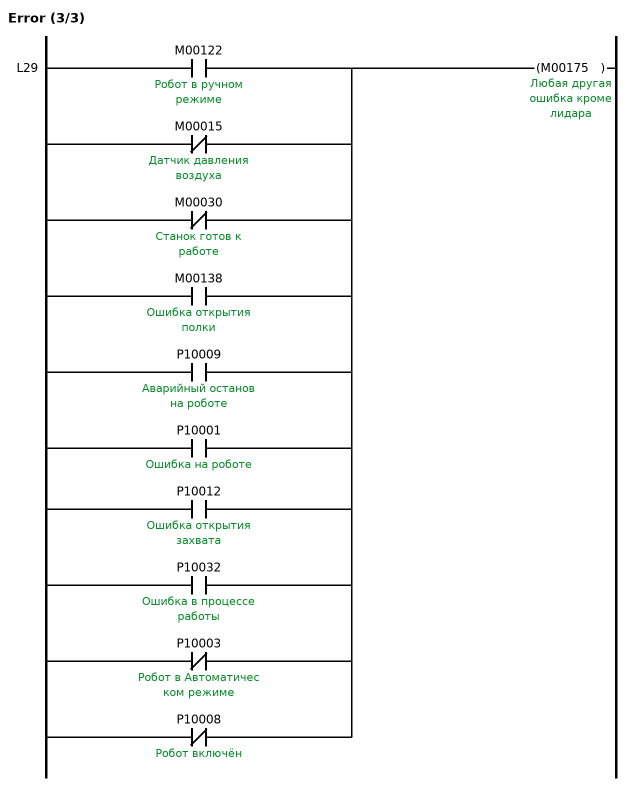
[picture p24: Error rungs L29-L29]
; L29
LOAD      M00122	// Робот в ручном режиме
OR NOT    M00015	// Датчик давления воздуха
OR NOT    M00030	// Станок готов к работе
OR        M00138	// Ошибка открытия полки
OR        P10009	// Аварийный останов на роботе
OR        P10001	// Ошибка на роботе
OR        P10012	// Ошибка открытия захвата
OR        P10032	// Ошибка в процессе работы
OR NOT    P10003	// Робот в Автоматическом режиме
OR NOT    P10008	// Робот включён
OUT       M00175	// Любая другая ошибка кроме лидара

PROGRAM Initialization (task: Scan Program)

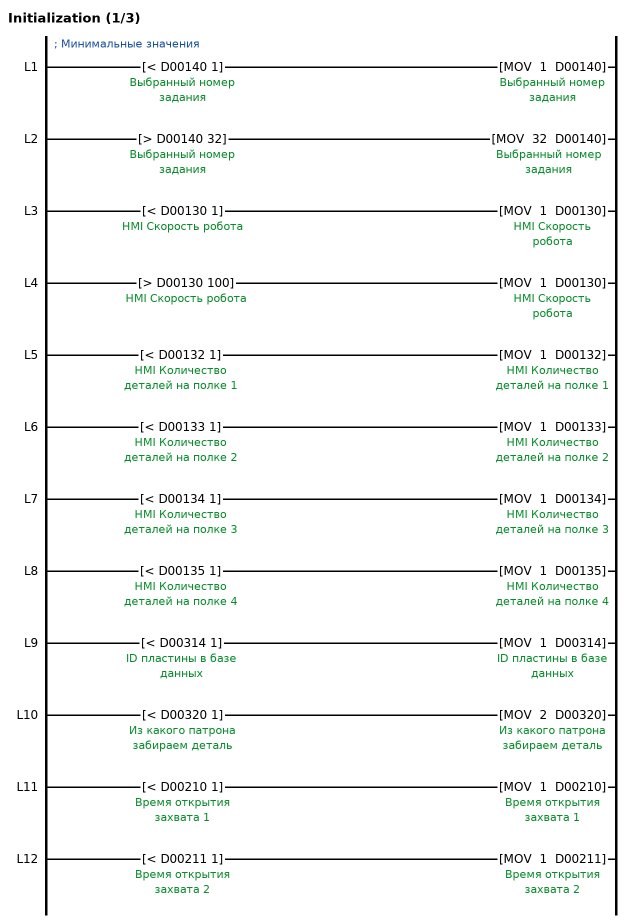
// Минимальные значения
; L1
LOAD<     D00140 1	// Выбранный номер задания
MOV       1 D00140	// Выбранный номер задания
; L2
LOAD>     D00140 32	// Выбранный номер задания
MOV       32 D00140	// Выбранный номер задания
; L3
LOAD<     D00130 1	// HMI Скорость робота
MOV       1 D00130	// HMI Скорость робота
; L4
LOAD>     D00130 100	// HMI Скорость робота
MOV       1 D00130	// HMI Скорость робота
; L5
LOAD<     D00132 1	// HMI Количество деталей на полке 1
MOV       1 D00132	// HMI Количество деталей на полке 1
; L6
LOAD<     D00133 1	// HMI Количество деталей на полке 2
MOV       1 D00133	// HMI Количество деталей на полке 2
; L7
LOAD<     D00134 1	// HMI Количество деталей на полке 3
MOV       1 D00134	// HMI Количество деталей на полке 3
; L8
LOAD<     D00135 1	// HMI Количество деталей на полке 4
MOV       1 D00135	// HMI Количество деталей на полке 4
; L9
LOAD<     D00314 1	// ID пластины в базе данных
MOV       1 D00314	// ID пластины в базе данных
; L10
LOAD<     D00320 1	// Из какого патрона забираем деталь
MOV       2 D00320	// Из какого патрона забираем деталь
; L11
LOAD<     D00210 1	// Время открытия захвата 1
MOV       1 D00210	// Время открытия захвата 1
; L12
LOAD<     D00211 1	// Время открытия захвата 2
MOV       1 D00211	// Время открытия захвата 2

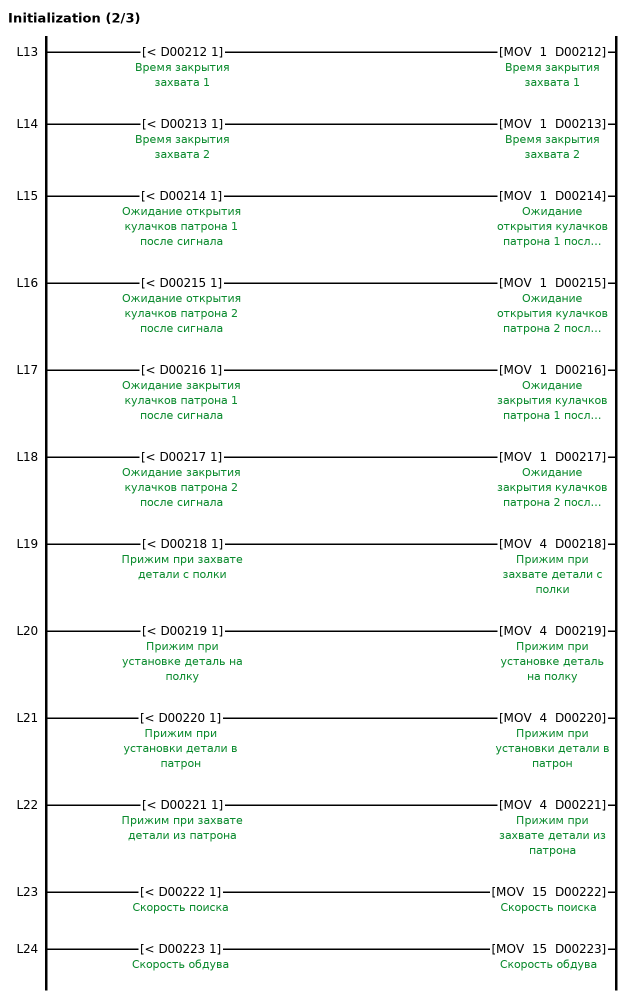
; L13
LOAD<     D00212 1	// Время закрытия захвата 1
MOV       1 D00212	// Время закрытия захвата 1
; L14
LOAD<     D00213 1	// Время закрытия захвата 2
MOV       1 D00213	// Время закрытия захвата 2
; L15
LOAD<     D00214 1	// Ожидание открытия кулачков патрона 1 после сигнала 
MOV       1 D00214	// Ожидание открытия кулачков патрона 1 после сигнала 
; L16
LOAD<     D00215 1	// Ожидание открытия кулачков патрона 2 после сигнала 
MOV       1 D00215	// Ожидание открытия кулачков патрона 2 после сигнала 
; L17
LOAD<     D00216 1	// Ожидание закрытия кулачков патрона 1 после сигнала 
MOV       1 D00216	// Ожидание закрытия кулачков патрона 1 после сигнала 
; L18
LOAD<     D00217 1	// Ожидание закрытия кулачков патрона 2 после сигнала 
MOV       1 D00217	// Ожидание закрытия кулачков патрона 2 после сигнала 
; L19
LOAD<     D00218 1	// Прижим при захвате детали с полки
MOV       4 D00218	// Прижим при захвате детали с полки
; L20
LOAD<     D00219 1	// Прижим при установке деталь на полку
MOV       4 D00219	// Прижим при установке деталь на полку
; L21
LOAD<     D00220 1	// Прижим при установки детали в патрон
MOV       4 D00220	// Прижим при установки детали в патрон
; L22
LOAD<     D00221 1	// Прижим при захвате детали из патрона
MOV       4 D00221	// Прижим при захвате детали из патрона
; L23
LOAD<     D00222 1	// Скорость поиска
MOV       15 D00222	// Скорость поиска
; L24
LOAD<     D00223 1	// Скорость обдува
MOV       15 D00223	// Скорость обдува

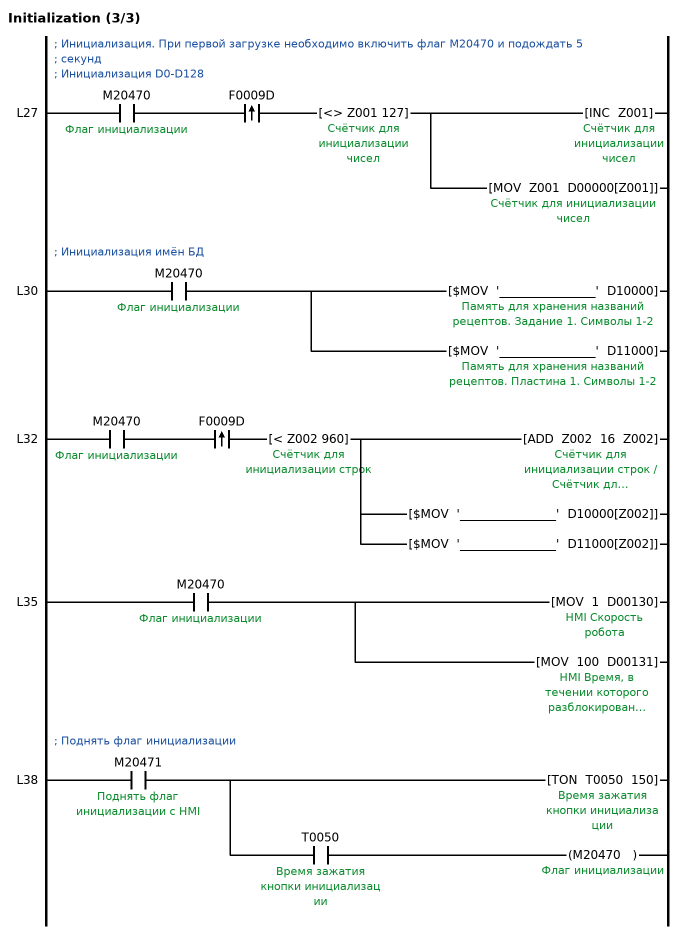
// Инициализация. При первой загрузке необходимо включить флаг M20470 и подождать 5 секунд
// Инициализация D0-D128
; L27
LOAD      M20470	// Флаг инициализации
ANDP      F0009D
AND<>     Z001 127	// Счётчик для инициализации чисел
INC       Z001	// Счётчик для инициализации чисел
MOV       Z001 D00000[Z001]	// Счётчик для инициализации чисел
// Инициализация имён БД
; L30
LOAD      M20470	// Флаг инициализации
$MOV      '________________' D10000	// Память для хранения названий рецептов. Задание 1. Символы 1-2
$MOV      '________________' D11000	// Память для хранения названий рецептов. Пластина 1. Символы 1-2
; L32
LOAD      M20470	// Флаг инициализации
ANDP      F0009D
AND<      Z002 960	// Счётчик для инициализации строк
ADD       Z002 16 Z002	// Счётчик для инициализации строк / Счётчик для инициализации строк
$MOV      '________________' D10000[Z002]
$MOV      '________________' D11000[Z002]
; L35
LOAD      M20470	// Флаг инициализации
MOV       1 D00130	// HMI Скорость робота
MOV       100 D00131	// HMI Время, в течении которого разблокирована полка после нажатия кнопки
// Поднять флаг инициализации
; L38
LOAD      M20471	// Поднять флаг инициализации с HMI
TON       T0050 150	// Время зажатия кнопки инициализации
AND       T0050	// Время зажатия кнопки инициализации
OUT       M20470	// Флаг инициализации

PROGRAM Shelves (task: Scan Program)

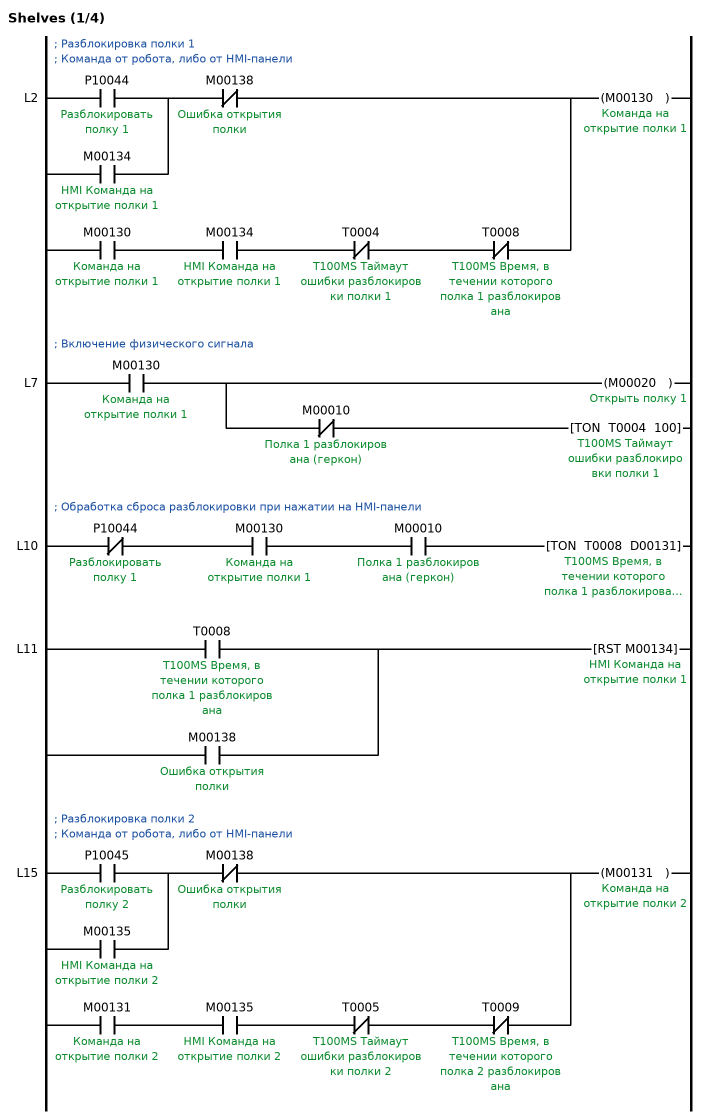
// Разблокировка полки 1
// Команда от робота, либо от HMI-панели
; L2
LOAD      P10044	// Разблокировать полку 1
OR        M00134	// HMI Команда на открытие полки 1
AND NOT   M00138	// Ошибка открытия полки
LOAD      M00130	// Команда на открытие полки 1
AND       M00134	// HMI Команда на открытие полки 1
AND NOT   T0004	// T100MS Таймаут ошибки разблокировки полки 1
AND NOT   T0008	// T100MS Время, в течении которого полка 1 разблокирована
OR LOAD
OUT       M00130	// Команда на открытие полки 1
// Включение физического сигнала
; L7
LOAD      M00130	// Команда на открытие полки 1
OUT       M00020	// Открыть полку 1
AND NOT   M00010	// Полка 1 разблокирована (геркон)
TON       T0004 100	// T100MS Таймаут ошибки разблокировки полки 1
// Обработка сброса разблокировки при нажатии на HMI-панели
; L10
LOAD NOT  P10044	// Разблокировать полку 1
AND       M00130	// Команда на открытие полки 1
AND       M00010	// Полка 1 разблокирована (геркон)
TON       T0008 D00131	// T100MS Время, в течении которого полка 1 разблокирована / HMI Время, в течении которого разблокирована полка после нажатия кнопки
; L11
LOAD      T0008	// T100MS Время, в течении которого полка 1 разблокирована
OR        M00138	// Ошибка открытия полки
RST       M00134	// HMI Команда на открытие полки 1
// Разблокировка полки 2
// Команда от робота, либо от HMI-панели
; L15
LOAD      P10045	// Разблокировать полку 2
OR        M00135	// HMI Команда на открытие полки 2
AND NOT   M00138	// Ошибка открытия полки
LOAD      M00131	// Команда на открытие полки 2
AND       M00135	// HMI Команда на открытие полки 2
AND NOT   T0005	// T100MS Таймаут ошибки разблокировки полки 2
AND NOT   T0009	// T100MS Время, в течении которого полка 2 разблокирована
OR LOAD
OUT       M00131	// Команда на открытие полки 2

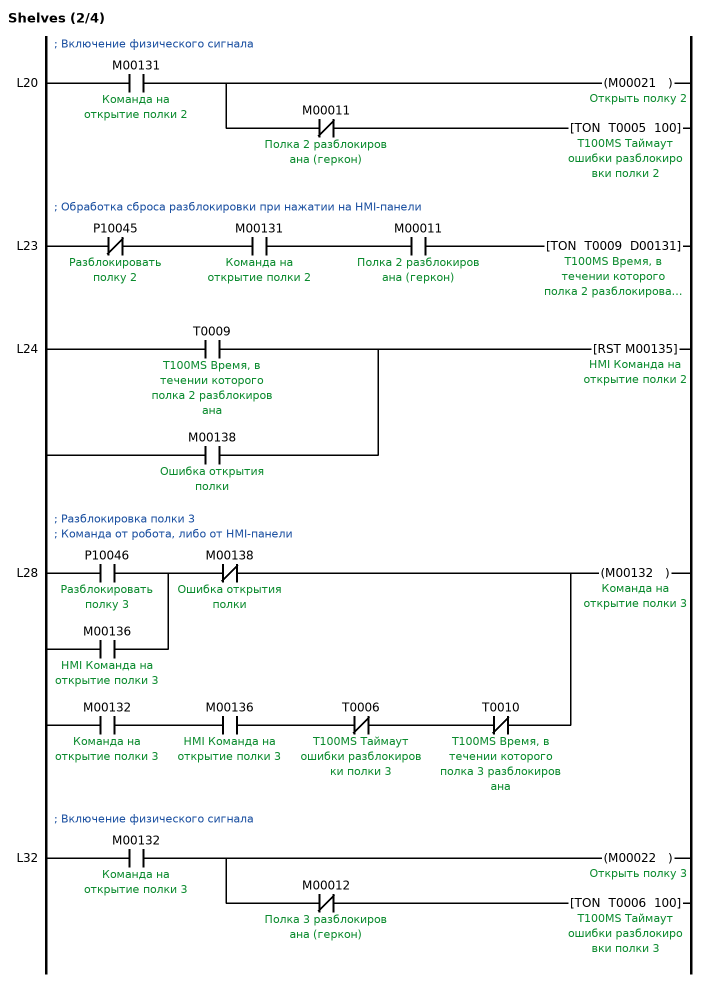
// Включение физического сигнала
; L20
LOAD      M00131	// Команда на открытие полки 2
OUT       M00021	// Открыть полку 2
AND NOT   M00011	// Полка 2 разблокирована (геркон)
TON       T0005 100	// T100MS Таймаут ошибки разблокировки полки 2
// Обработка сброса разблокировки при нажатии на HMI-панели
; L23
LOAD NOT  P10045	// Разблокировать полку 2
AND       M00131	// Команда на открытие полки 2
AND       M00011	// Полка 2 разблокирована (геркон)
TON       T0009 D00131	// T100MS Время, в течении которого полка 2 разблокирована / HMI Время, в течении которого разблокирована полка после нажатия кнопки
; L24
LOAD      T0009	// T100MS Время, в течении которого полка 2 разблокирована
OR        M00138	// Ошибка открытия полки
RST       M00135	// HMI Команда на открытие полки 2
// Разблокировка полки 3
// Команда от робота, либо от HMI-панели
; L28
LOAD      P10046	// Разблокировать полку 3
OR        M00136	// HMI Команда на открытие полки 3
AND NOT   M00138	// Ошибка открытия полки
LOAD      M00132	// Команда на открытие полки 3
AND       M00136	// HMI Команда на открытие полки 3
AND NOT   T0006	// T100MS Таймаут ошибки разблокировки полки 3
AND NOT   T0010	// T100MS Время, в течении которого полка 3 разблокирована
OR LOAD
OUT       M00132	// Команда на открытие полки 3
// Включение физического сигнала
; L32
LOAD      M00132	// Команда на открытие полки 3
OUT       M00022	// Открыть полку 3
AND NOT   M00012	// Полка 3 разблокирована (геркон)
TON       T0006 100	// T100MS Таймаут ошибки разблокировки полки 3

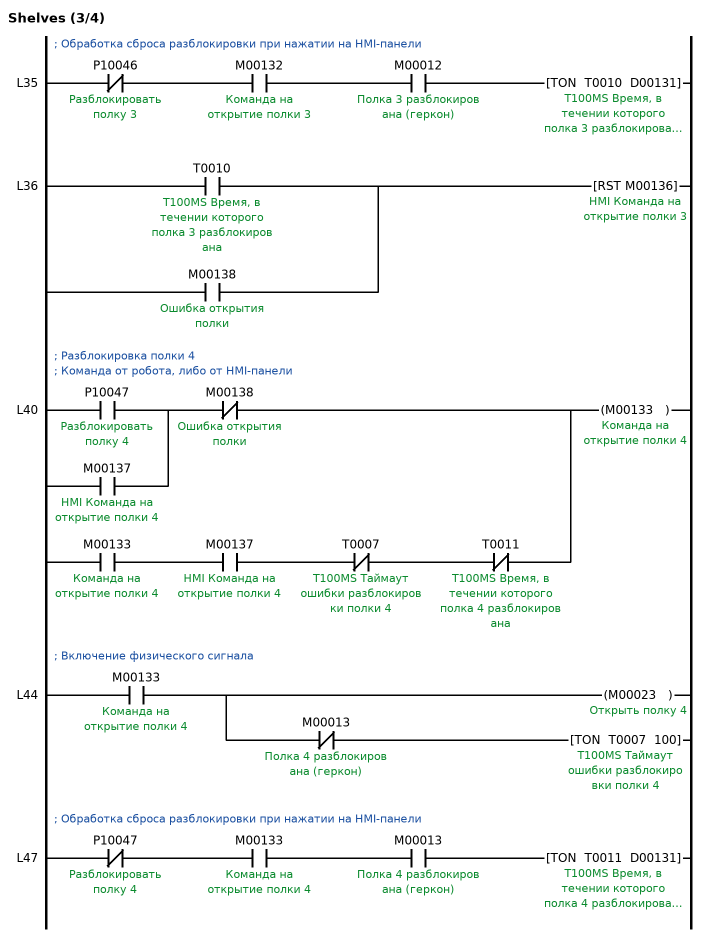
// Обработка сброса разблокировки при нажатии на HMI-панели
; L35
LOAD NOT  P10046	// Разблокировать полку 3
AND       M00132	// Команда на открытие полки 3
AND       M00012	// Полка 3 разблокирована (геркон)
TON       T0010 D00131	// T100MS Время, в течении которого полка 3 разблокирована / HMI Время, в течении которого разблокирована полка после нажатия кнопки
; L36
LOAD      T0010	// T100MS Время, в течении которого полка 3 разблокирована
OR        M00138	// Ошибка открытия полки
RST       M00136	// HMI Команда на открытие полки 3
// Разблокировка полки 4
// Команда от робота, либо от HMI-панели
; L40
LOAD      P10047	// Разблокировать полку 4
OR        M00137	// HMI Команда на открытие полки 4
AND NOT   M00138	// Ошибка открытия полки
LOAD      M00133	// Команда на открытие полки 4
AND       M00137	// HMI Команда на открытие полки 4
AND NOT   T0007	// T100MS Таймаут ошибки разблокировки полки 4
AND NOT   T0011	// T100MS Время, в течении которого полка 4 разблокирована
OR LOAD
OUT       M00133	// Команда на открытие полки 4
// Включение физического сигнала
; L44
LOAD      M00133	// Команда на открытие полки 4
OUT       M00023	// Открыть полку 4
AND NOT   M00013	// Полка 4 разблокирована (геркон)
TON       T0007 100	// T100MS Таймаут ошибки разблокировки полки 4
// Обработка сброса разблокировки при нажатии на HMI-панели
; L47
LOAD NOT  P10047	// Разблокировать полку 4
AND       M00133	// Команда на открытие полки 4
AND       M00013	// Полка 4 разблокирована (геркон)
TON       T0011 D00131	// T100MS Время, в течении которого полка 4 разблокирована / HMI Время, в течении которого разблокирована полка после нажатия кнопки

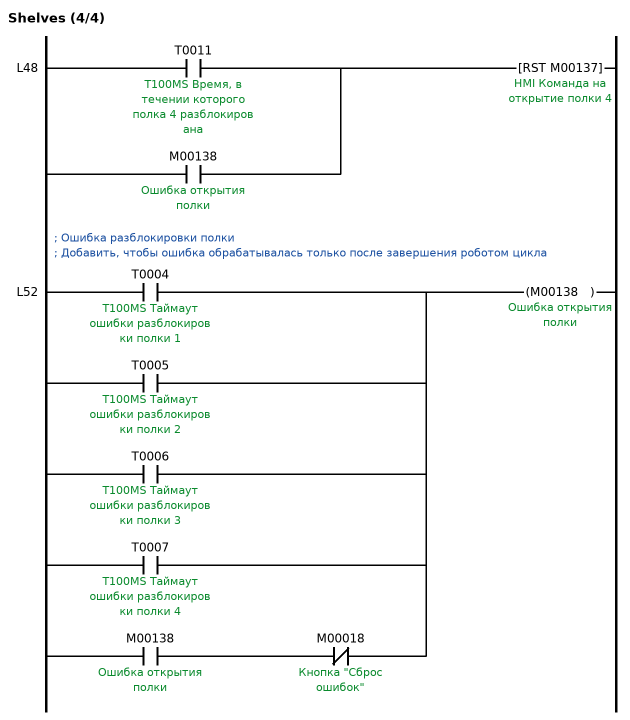
; L48
LOAD      T0011	// T100MS Время, в течении которого полка 4 разблокирована
OR        M00138	// Ошибка открытия полки
RST       M00137	// HMI Команда на открытие полки 4
// Ошибка разблокировки полки
// Добавить, чтобы ошибка обрабатывалась только после завершения роботом цикла
; L52
LOAD      T0004	// T100MS Таймаут ошибки разблокировки полки 1
OR        T0005	// T100MS Таймаут ошибки разблокировки полки 2
OR        T0006	// T100MS Таймаут ошибки разблокировки полки 3
OR        T0007	// T100MS Таймаут ошибки разблокировки полки 4
LOAD      M00138	// Ошибка открытия полки
AND NOT   M00018	// Кнопка "Сброс ошибок"
OR LOAD
OUT       M00138	// Ошибка открытия полки

PROGRAM Database (task: Scan Program)

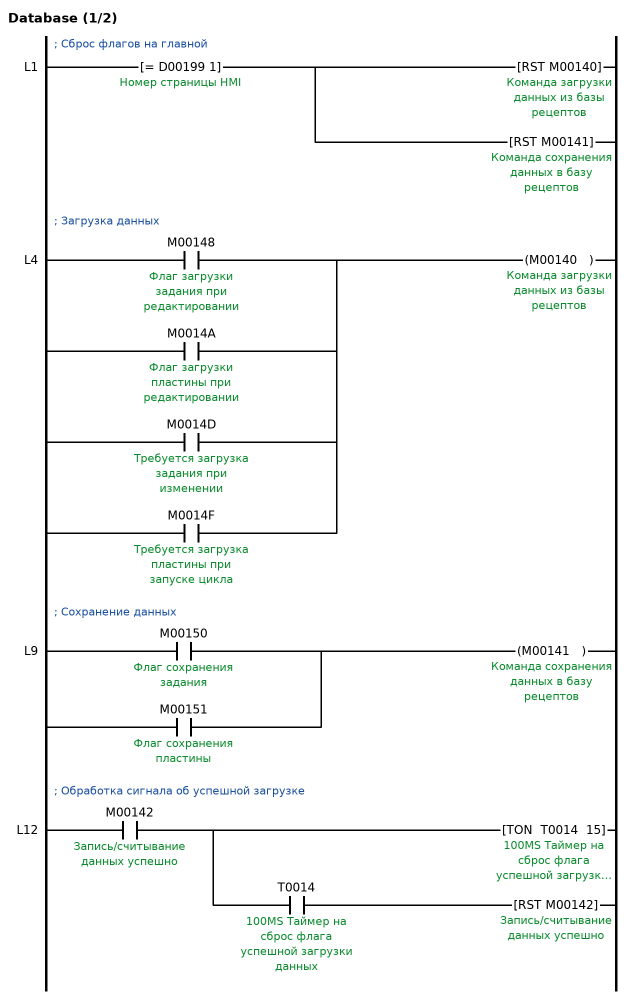
// Сброс флагов на главной
; L1
LOAD=     D00199 1	// Номер страницы HMI
RST       M00140	// Команда загрузки данных из базы рецептов
RST       M00141	// Команда сохранения данных в базу рецептов
// Загрузка данных
; L4
LOAD      M00148	// Флаг загрузки задания при редактировании
OR        M0014A	// Флаг загрузки пластины при редактировании
OR        M0014D	// Требуется загрузка задания при изменении
OR        M0014F	// Требуется загрузка пластины при запуске цикла
OUT       M00140	// Команда загрузки данных из базы рецептов
// Сохранение данных
; L9
LOAD      M00150	// Флаг сохранения задания
OR        M00151	// Флаг сохранения пластины
OUT       M00141	// Команда сохранения данных в базу рецептов
// Обработка сигнала об успешной загрузке
; L12
LOAD      M00142	// Запись/считывание данных успешно
TON       T0014 15	// 100MS Таймер на сброс флага успешной загрузки данных
AND       T0014	// 100MS Таймер на сброс флага успешной загрузки данных
RST       M00142	// Запись/считывание данных успешно

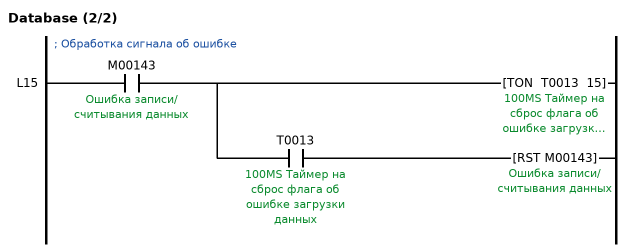
// Обработка сигнала об ошибке
; L15
LOAD      M00143	// Ошибка записи/считывания данных
TON       T0013 15	// 100MS Таймер на сброс флага об ошибке загрузки данных
AND       T0013	// 100MS Таймер на сброс флага об ошибке загрузки данных
RST       M00143	// Ошибка записи/считывания данных

PROGRAM HMI (task: Scan Program)

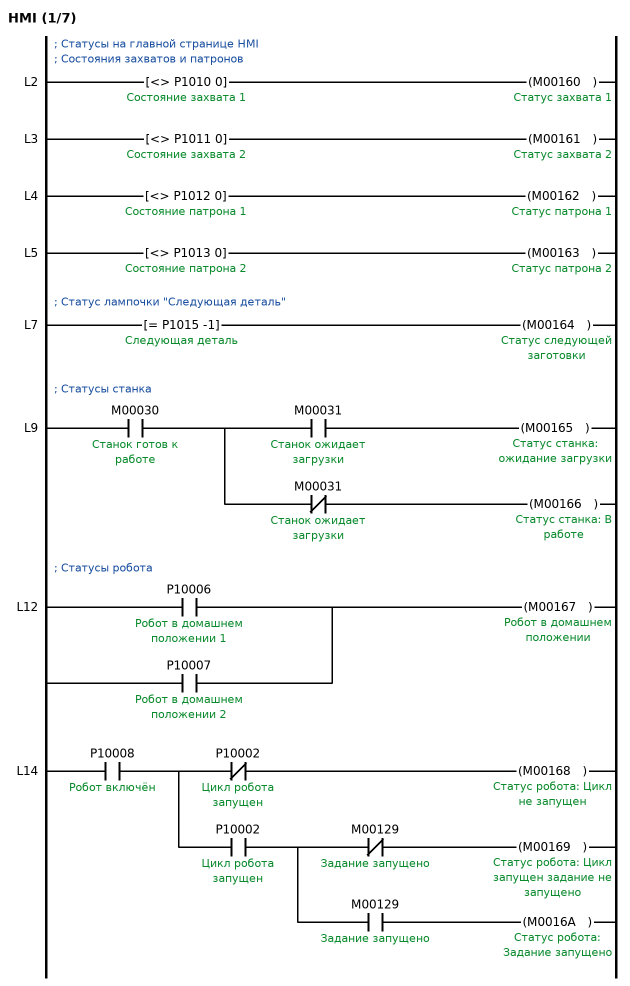
// Статусы на главной странице HMI
// Состояния захватов и патронов
; L2
LOAD<>    P1010 0	// Состояние захвата 1
OUT       M00160	// Статус захвата 1
; L3
LOAD<>    P1011 0	// Состояние захвата 2
OUT       M00161	// Статус захвата 2
; L4
LOAD<>    P1012 0	// Состояние патрона 1
OUT       M00162	// Статус патрона 1
; L5
LOAD<>    P1013 0	// Состояние патрона 2
OUT       M00163	// Статус патрона 2
// Статус лампочки "Следующая деталь"
; L7
LOAD=     P1015 -1	// Следующая деталь
OUT       M00164	// Статус следующей заготовки 
// Статусы станка
; L9
LOAD      M00030	// Станок готов к работе
MPUSH
AND       M00031	// Станок ожидает загрузки
OUT       M00165	// Статус станка: ожидание загрузки
MPOP
AND NOT   M00031	// Станок ожидает загрузки
OUT       M00166	// Статус станка: В работе
// Статусы робота
; L12
LOAD      P10006	// Робот в домашнем положении 1
OR        P10007	// Робот в домашнем положении 2
OUT       M00167	// Робот в домашнем положении
; L14
LOAD      P10008	// Робот включён
MPUSH
AND NOT   P10002	// Цикл робота запущен
OUT       M00168	// Статус робота: Цикл не запущен
MPOP
AND       P10002	// Цикл робота запущен
MPUSH
AND NOT   M00129	// Задание запущено
OUT       M00169	// Статус робота: Цикл запущен задание не запущено
MPOP
AND       M00129	// Задание запущено
OUT       M0016A	// Статус робота: Задание запущено

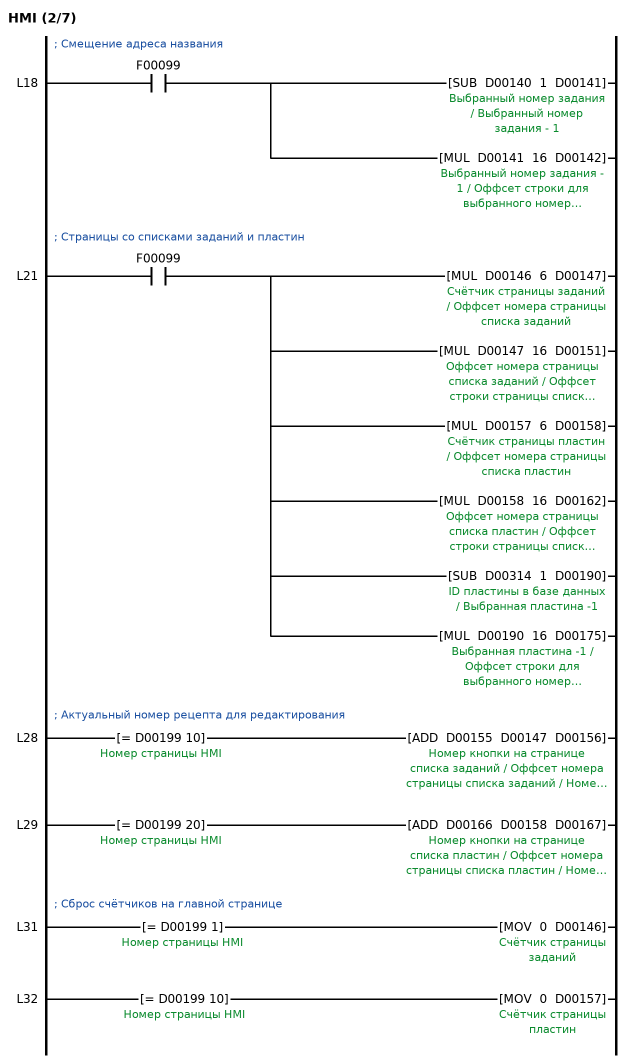
// Смещение адреса названия
; L18
LOAD      F00099
SUB       D00140 1 D00141	// Выбранный номер задания / Выбранный номер задания - 1
MUL       D00141 16 D00142	// Выбранный номер задания - 1 / Оффсет строки для выбранного номера названия
// Страницы со списками заданий и пластин
; L21
LOAD      F00099
MUL       D00146 6 D00147	// Счётчик страницы заданий / Оффсет номера страницы списка заданий
MUL       D00147 16 D00151	// Оффсет номера страницы списка заданий / Оффсет строки страницы списка заданий
MUL       D00157 6 D00158	// Счётчик страницы пластин / Оффсет номера страницы списка пластин
MUL       D00158 16 D00162	// Оффсет номера страницы списка пластин / Оффсет строки страницы списка пластин
SUB       D00314 1 D00190	// ID пластины в базе данных / Выбранная пластина -1
MUL       D00190 16 D00175	// Выбранная пластина -1 / Оффсет строки для выбранного номера пластины
// Актуальный номер рецепта для редактирования
; L28
LOAD=     D00199 10	// Номер страницы HMI
ADD       D00155 D00147 D00156	// Номер кнопки на странице списка заданий / Оффсет номера страницы списка заданий / Номер редактируемого задания
; L29
LOAD=     D00199 20	// Номер страницы HMI
ADD       D00166 D00158 D00167	// Номер кнопки на странице списка пластин / Оффсет номера страницы списка пластин / Номер редактируемой пластины
// Сброс счётчиков на главной странице
; L31
LOAD=     D00199 1	// Номер страницы HMI
MOV       0 D00146	// Счётчик страницы заданий
; L32
LOAD=     D00199 10	// Номер страницы HMI
MOV       0 D00157	// Счётчик страницы пластин

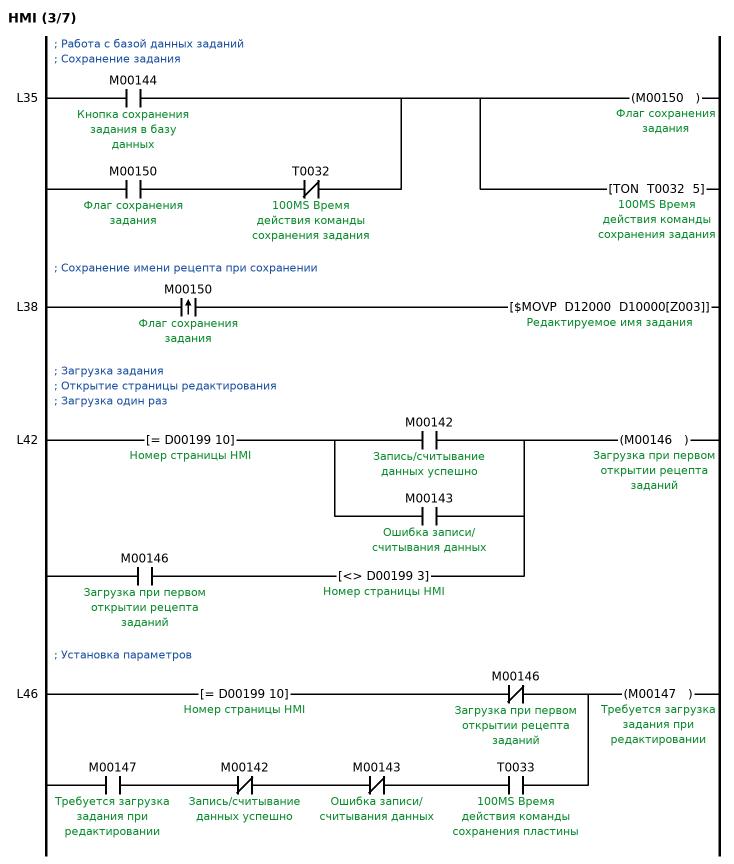
// Работа с базой данных заданий
// Сохранение задания
; L35
LOAD      M00144	// Кнопка сохранения задания в базу данных
LOAD      M00150	// Флаг сохранения задания
AND NOT   T0032	// 100MS Время действия команды сохранения задания
OR LOAD
OUT       M00150	// Флаг сохранения задания
TON       T0032 5	// 100MS Время действия команды сохранения задания
// Сохранение имени рецепта при сохранении
; L38
LOADP     M00150	// Флаг сохранения задания
$MOVP     D12000 D10000[Z003]	// Редактируемое имя задания
// Загрузка задания
// Открытие страницы редактирования
// Загрузка один раз
; L42
LOAD=     D00199 10	// Номер страницы HMI
LOAD      M00142	// Запись/считывание данных успешно
OR        M00143	// Ошибка записи/считывания данных
AND LOAD
LOAD      M00146	// Загрузка при первом открытии рецепта заданий
AND<>     D00199 3	// Номер страницы HMI
OR LOAD
OUT       M00146	// Загрузка при первом открытии рецепта заданий
// Установка параметров
; L46
LOAD=     D00199 10	// Номер страницы HMI
AND NOT   M00146	// Загрузка при первом открытии рецепта заданий
LOAD      M00147	// Требуется загрузка задания при редактировании
AND NOT   M00142	// Запись/считывание данных успешно
AND NOT   M00143	// Ошибка записи/считывания данных
AND       T0033	// 100MS Время действия команды сохранения пластины
OR LOAD
OUT       M00147	// Требуется загрузка задания при редактировании

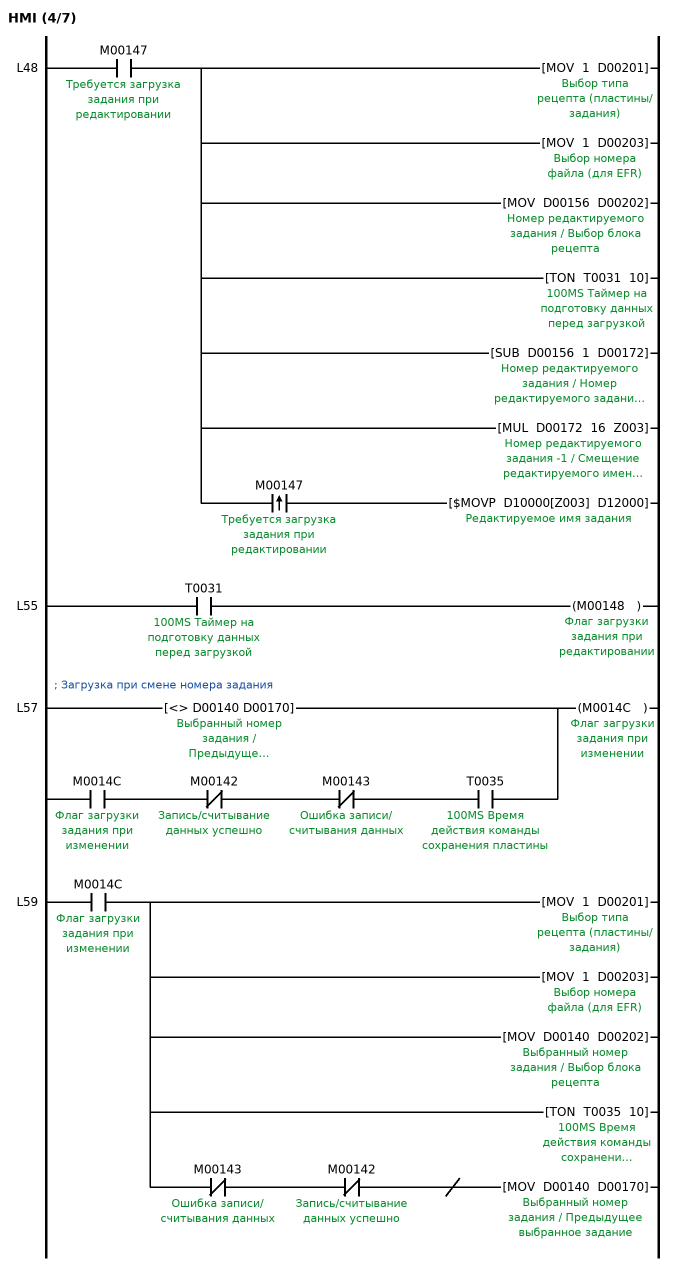
; L48
LOAD      M00147	// Требуется загрузка задания при редактировании
MOV       1 D00201	// Выбор типа рецепта (пластины/задания)
MOV       1 D00203	// Выбор номера файла (для EFR)
MOV       D00156 D00202	// Номер редактируемого задания / Выбор блока рецепта
TON       T0031 10	// 100MS Таймер на подготовку данных перед загрузкой
SUB       D00156 1 D00172	// Номер редактируемого задания / Номер редактируемого задания -1
MUL       D00172 16 Z003	// Номер редактируемого задания -1 / Смещение редактируемого имени задания
ANDP      M00147	// Требуется загрузка задания при редактировании
$MOVP     D10000[Z003] D12000	// Редактируемое имя задания
; L55
LOAD      T0031	// 100MS Таймер на подготовку данных перед загрузкой
OUT       M00148	// Флаг загрузки задания при редактировании
// Загрузка при смене номера задания
; L57
LOAD<>    D00140 D00170	// Выбранный номер задания / Предыдущее выбранное задание
LOAD      M0014C	// Флаг загрузки задания при изменении
AND NOT   M00142	// Запись/считывание данных успешно
AND NOT   M00143	// Ошибка записи/считывания данных
AND       T0035	// 100MS Время действия команды сохранения пластины
OR LOAD
OUT       M0014C	// Флаг загрузки задания при изменении
; L59
LOAD      M0014C	// Флаг загрузки задания при изменении
MOV       1 D00201	// Выбор типа рецепта (пластины/задания)
MOV       1 D00203	// Выбор номера файла (для EFR)
MOV       D00140 D00202	// Выбранный номер задания / Выбор блока рецепта
TON       T0035 10	// 100MS Время действия команды сохранения пластины
AND NOT   M00143	// Ошибка записи/считывания данных
AND NOT   M00142	// Запись/считывание данных успешно
NOT
MOV       D00140 D00170	// Выбранный номер задания / Предыдущее выбранное задание

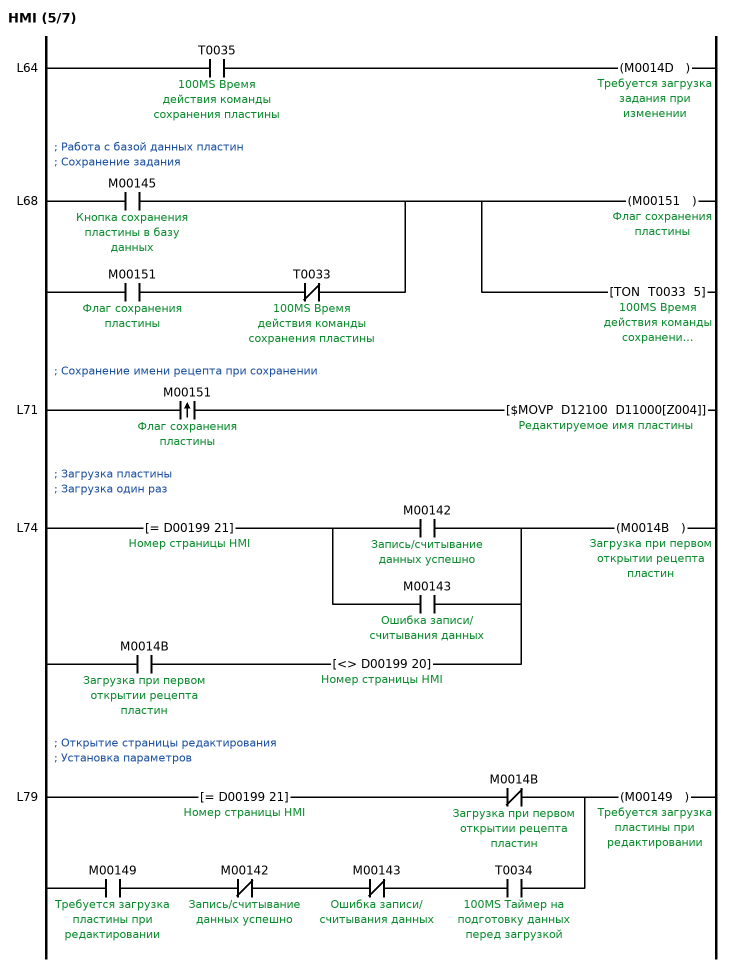
; L64
LOAD      T0035	// 100MS Время действия команды сохранения пластины
OUT       M0014D	// Требуется загрузка задания при изменении
//  
// Работа с базой данных пластин
// Сохранение задания
; L68
LOAD      M00145	// Кнопка сохранения пластины в базу данных
LOAD      M00151	// Флаг сохранения пластины
AND NOT   T0033	// 100MS Время действия команды сохранения пластины
OR LOAD
OUT       M00151	// Флаг сохранения пластины
TON       T0033 5	// 100MS Время действия команды сохранения пластины
// Сохранение имени рецепта при сохранении
; L71
LOADP     M00151	// Флаг сохранения пластины
$MOVP     D12100 D11000[Z004]	// Редактируемое имя пластины
// Загрузка пластины
// Загрузка один раз
; L74
LOAD=     D00199 21	// Номер страницы HMI
LOAD      M00142	// Запись/считывание данных успешно
OR        M00143	// Ошибка записи/считывания данных
AND LOAD
LOAD      M0014B	// Загрузка при первом открытии рецепта пластин
AND<>     D00199 20	// Номер страницы HMI
OR LOAD
OUT       M0014B	// Загрузка при первом открытии рецепта пластин
// Открытие страницы редактирования
// Установка параметров
; L79
LOAD=     D00199 21	// Номер страницы HMI
AND NOT   M0014B	// Загрузка при первом открытии рецепта пластин
LOAD      M00149	// Требуется загрузка пластины при редактировании
AND NOT   M00142	// Запись/считывание данных успешно
AND NOT   M00143	// Ошибка записи/считывания данных
AND       T0034	// 100MS Таймер на подготовку данных перед загрузкой
OR LOAD
OUT       M00149	// Требуется загрузка пластины при редактировании

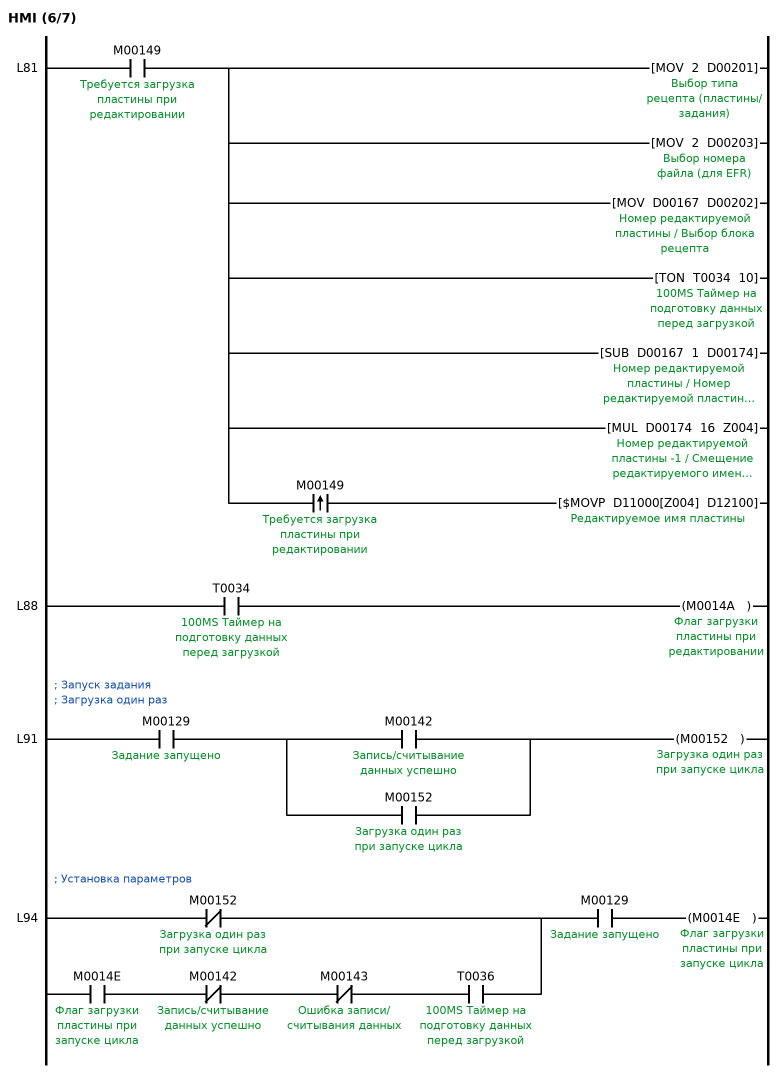
; L81
LOAD      M00149	// Требуется загрузка пластины при редактировании
MOV       2 D00201	// Выбор типа рецепта (пластины/задания)
MOV       2 D00203	// Выбор номера файла (для EFR)
MOV       D00167 D00202	// Номер редактируемой пластины / Выбор блока рецепта
TON       T0034 10	// 100MS Таймер на подготовку данных перед загрузкой
SUB       D00167 1 D00174	// Номер редактируемой пластины / Номер редактируемой пластины -1
MUL       D00174 16 Z004	// Номер редактируемой пластины -1 / Смещение редактируемого имени пластины
ANDP      M00149	// Требуется загрузка пластины при редактировании
$MOVP     D11000[Z004] D12100	// Редактируемое имя пластины
; L88
LOAD      T0034	// 100MS Таймер на подготовку данных перед загрузкой
OUT       M0014A	// Флаг загрузки пластины при редактировании
// Запуск задания
// Загрузка один раз
; L91
LOAD      M00129	// Задание запущено
LOAD      M00142	// Запись/считывание данных успешно
OR        M00152	// Загрузка один раз при запуске цикла
AND LOAD
OUT       M00152	// Загрузка один раз при запуске цикла
// Установка параметров
; L94
LOAD NOT  M00152	// Загрузка один раз при запуске цикла
LOAD      M0014E	// Флаг загрузки пластины при запуске цикла
AND NOT   M00142	// Запись/считывание данных успешно
AND NOT   M00143	// Ошибка записи/считывания данных
AND       T0036	// 100MS Таймер на подготовку данных перед загрузкой
OR LOAD
AND       M00129	// Задание запущено
OUT       M0014E	// Флаг загрузки пластины при запуске цикла

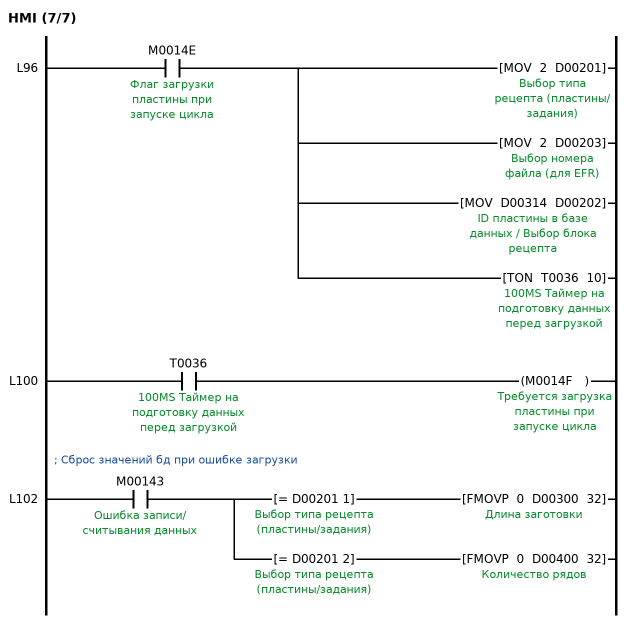
; L96
LOAD      M0014E	// Флаг загрузки пластины при запуске цикла
MOV       2 D00201	// Выбор типа рецепта (пластины/задания)
MOV       2 D00203	// Выбор номера файла (для EFR)
MOV       D00314 D00202	// ID пластины в базе данных / Выбор блока рецепта
TON       T0036 10	// 100MS Таймер на подготовку данных перед загрузкой
; L100
LOAD      T0036	// 100MS Таймер на подготовку данных перед загрузкой
OUT       M0014F	// Требуется загрузка пластины при запуске цикла
// Сброс значений бд при ошибке загрузки
; L102
LOAD      M00143	// Ошибка записи/считывания данных
MPUSH
AND=      D00201 1	// Выбор типа рецепта (пластины/задания)
FMOVP     0 D00300 32	// Длина заготовки
MPOP
AND=      D00201 2	// Выбор типа рецепта (пластины/задания)
FMOVP     0 D00400 32	// Количество рядов

VARIABLES AND COMMENTS (devices not used above)
P1000C	BIT	Требуется замена батареи питания энкодера
D00000	WORD	Фиксированное число 0
D00001	WORD	Фиксированное число 1
D00002	WORD	Фиксированное число 2
D00003	WORD	Фиксированное число 3
D00004	WORD	Фиксированное число 4
D00005	WORD	Фиксированное число 5
D00006	WORD	Фиксированное число 6
D00007	WORD	Фиксированное число 7
D00008	WORD	Фиксированное число 8
D00009	WORD	Фиксированное число 9
D00010	WORD	Фиксированное число 10
D00011	WORD	Фиксированное число 11
D00012	WORD	Фиксированное число 12
D00013	WORD	Фиксированное число 13
D00014	WORD	Фиксированное число 14
D00015	WORD	Фиксированное число 15
D00016	WORD	Фиксированное число 16
D00017	WORD	Фиксированное число 17
D00018	WORD	Фиксированное число 18
D00019	WORD	Фиксированное число 19
D00020	WORD	Фиксированное число 20
D00021	WORD	Фиксированное число 21
D00022	WORD	Фиксированное число 22
D00023	WORD	Фиксированное число 23
D00024	WORD	Фиксированное число 24
D00025	WORD	Фиксированное число 25
D00026	WORD	Фиксированное число 26
D00027	WORD	Фиксированное число 27
D00028	WORD	Фиксированное число 28
D00029	WORD	Фиксированное число 29
D00030	WORD	Фиксированное число 30
D00031	WORD	Фиксированное число 31
D00032	WORD	Фиксированное число 32
D00033	WORD	Фиксированное число 33
D00034	WORD	Фиксированное число 34
D00035	WORD	Фиксированное число 35
D00036	WORD	Фиксированное число 36
D00037	WORD	Фиксированное число 37
D00038	WORD	Фиксированное число 38
D00039	WORD	Фиксированное число 39
D00040	WORD	Фиксированное число 40
D00041	WORD	Фиксированное число 41
D00042	WORD	Фиксированное число 42
D00043	WORD	Фиксированное число 43
D00044	WORD	Фиксированное число 44
D00045	WORD	Фиксированное число 45
D00046	WORD	Фиксированное число 46
D00047	WORD	Фиксированное число 47
D00048	WORD	Фиксированное число 48
D00049	WORD	Фиксированное число 49
D00050	WORD	Фиксированное число 50
D00051	WORD	Фиксированное число 51
D00052	WORD	Фиксированное число 52
D00053	WORD	Фиксированное число 53
D00054	WORD	Фиксированное число 54
D00055	WORD	Фиксированное число 55
D00056	WORD	Фиксированное число 56
D00057	WORD	Фиксированное число 57
D00058	WORD	Фиксированное число 58
D00059	WORD	Фиксированное число 59
D00060	WORD	Фиксированное число 60
D00061	WORD	Фиксированное число 61
D00062	WORD	Фиксированное число 62
D00063	WORD	Фиксированное число 63
D00064	WORD	Фиксированное число 64
D00065	WORD	Фиксированное число 65
D00066	WORD	Фиксированное число 66
D00067	WORD	Фиксированное число 67
D00068	WORD	Фиксированное число 68
D00069	WORD	Фиксированное число 69
D00070	WORD	Фиксированное число 70
D00071	WORD	Фиксированное число 71
D00072	WORD	Фиксированное число 72
D00073	WORD	Фиксированное число 73
D00074	WORD	Фиксированное число 74
D00075	WORD	Фиксированное число 75
D00076	WORD	Фиксированное число 76
D00077	WORD	Фиксированное число 77
D00078	WORD	Фиксированное число 78
D00079	WORD	Фиксированное число 79
D00080	WORD	Фиксированное число 80
D00081	WORD	Фиксированное число 81
D00082	WORD	Фиксированное число 82
D00083	WORD	Фиксированное число 83
D00084	WORD	Фиксированное число 84
D00085	WORD	Фиксированное число 85
D00086	WORD	Фиксированное число 86
D00087	WORD	Фиксированное число 87
D00088	WORD	Фиксированное число 88
D00089	WORD	Фиксированное число 89
D00090	WORD	Фиксированное число 90
D00091	WORD	Фиксированное число 91
D00092	WORD	Фиксированное число 92
D00093	WORD	Фиксированное число 93
D00094	WORD	Фиксированное число 94
D00095	WORD	Фиксированное число 95
D00096	WORD	Фиксированное число 96
D00097	WORD	Фиксированное число 97
D00098	WORD	Фиксированное число 98
D00099	WORD	Фиксированное число 99
D00100	WORD	Фиксированное число 100
D00101	WORD	Фиксированное число 101
D00102	WORD	Фиксированное число 102
D00103	WORD	Фиксированное число 103
D00104	WORD	Фиксированное число 104
D00105	WORD	Фиксированное число 105
D00106	WORD	Фиксированное число 106
D00107	WORD	Фиксированное число 107
D00108	WORD	Фиксированное число 108
D00109	WORD	Фиксированное число 109
D00110	WORD	Фиксированное число 110
D00111	WORD	Фиксированное число 111
D00112	WORD	Фиксированное число 112
D00113	WORD	Фиксированное число 113
D00114	WORD	Фиксированное число 114
D00115	WORD	Фиксированное число 115
D00116	WORD	Фиксированное число 116
D00117	WORD	Фиксированное число 117
D00118	WORD	Фиксированное число 118
D00119	WORD	Фиксированное число 119
D00120	WORD	Фиксированное число 120
D00121	WORD	Фиксированное число 121
D00122	WORD	Фиксированное число 122
D00123	WORD	Фиксированное число 123
D00124	WORD	Фиксированное число 124
D00125	WORD	Фиксированное число 125
D00126	WORD	Фиксированное число 126
D00127	WORD	Фиксированное число 127
D00128	WORD	Фиксированное число 128
P10010	BIT	Захват 1 открыт
P10011	BIT	Захват 2 открыт
P10013	BIT	Захват 1 датчик сработал
P10014	BIT	Захват 2 датчик сработал
P10030	BIT	Робот готов к запуску задания
P11010	BIT	Открыть захват 1
P11011	BIT	Закрыть захват 1
P11012	BIT	Открыть захват 2
P11013	BIT	Закрыть захват 2
M00139	BIT	Индикатор ошибки открытия полки
P10037	BIT	Данные считаны
P10040	BIT	Полка 1 открыта
P10041	BIT	Полка 2 открыта
P10042	BIT	Полка 3 открыта
P10043	BIT	Полка 4 открыта
P10100	BIT	Состояние захвата 1
P10110	BIT	Состояние захвата 2
P10120	BIT	Состояние патрона 1
P10130	BIT	Состояние патрона 2
P10140	BIT	Обработано деталей
P11100	BIT	Скорость робота
P1014	WORD	Обработано деталей
P1136E	BIT	Реверс захвата 2
P1136F	BIT	Реверс захвата 1
P11374	BIT	В какой патрон ставим заготовку
P11376	BIT	Каким захватом берём заготовку
P11380	BIT	Смещение первого ряда относительно нуля Y
P11390	BIT	Смещение первого ряда относительно нуля Х
P11400	BIT	Смещение чётного ряда
P11410	BIT	Расстояние между ячейками
P11420	BIT	Расстояние между рядами
P11450	BIT	Тело кулачков в Патроне 2
P11460	BIT	Высота кулачков в Патроне 2
P11470	BIT	Тело кулачков в Патроне 1
P11480	BIT	Высота кулачков в Патроне 1
P11490	BIT	Тело кулачков в захвате 2
P11500	BIT	Высота кулачков в захвате 2
P11510	BIT	Тело кулачков в захвате 1
P11520	BIT	Высота кулачков в захвате 1
P11530	BIT	Длина полуфабриката
P11540	BIT	Длина детали
P11550	BIT	Длина заготовки
D00200	WORD	Код ошибки работы с базой данных
D00323	WORD	Параметры рецептов Пластин
D00324	WORD	Параметры рецептов Пластин
D00325	WORD	Параметры рецептов Пластин
D00326	WORD	Параметры рецептов Пластин
D00327	WORD	Параметры рецептов Пластин
D00328	WORD	Параметры рецептов Пластин
D00329	WORD	Параметры рецептов Пластин
D00330	WORD	Параметры рецептов Пластин
D00331	WORD	Параметры рецептов Пластин
D00332	WORD	Параметры рецептов Пластин
D00333	WORD	Параметры рецептов Пластин
D00334	WORD	Параметры рецептов Пластин
D00335	WORD	Параметры рецептов Пластин
D00336	WORD	Параметры рецептов Пластин
D00337	WORD	Параметры рецептов Пластин
D00338	WORD	Параметры рецептов Пластин
D00339	WORD	Параметры рецептов Пластин
D00340	WORD	Параметры рецептов Пластин
D00341	WORD	Параметры рецептов Пластин
D00342	WORD	Параметры рецептов Пластин
D00343	WORD	Параметры рецептов Пластин
D00344	WORD	Параметры рецептов Пластин
D00345	WORD	Параметры рецептов Пластин
D00346	WORD	Параметры рецептов Пластин
D00347	WORD	Параметры рецептов Пластин
D00348	WORD	Параметры рецептов Пластин
D00349	WORD	Параметры рецептов Пластин
D00350	WORD	Параметры рецептов Пластин
D00351	WORD	Параметры рецептов Пластин
D00352	WORD	Параметры рецептов Пластин
D00353	WORD	Параметры рецептов Пластин
D00354	WORD	Параметры рецептов Пластин
D00355	WORD	Параметры рецептов Пластин
D00356	WORD	Параметры рецептов Пластин
D00357	WORD	Параметры рецептов Пластин
D00358	WORD	Параметры рецептов Пластин
D00359	WORD	Параметры рецептов Пластин
D00360	WORD	Параметры рецептов Пластин
D00361	WORD	Параметры рецептов Пластин
D00362	WORD	Параметры рецептов Пластин
D00363	WORD	Параметры рецептов Пластин
D00364	WORD	Параметры рецептов Пластин
D00365	WORD	Параметры рецептов Пластин
D00366	WORD	Параметры рецептов Пластин
D00367	WORD	Параметры рецептов Пластин
D00368	WORD	Параметры рецептов Пластин
D00369	WORD	Параметры рецептов Пластин
D00370	WORD	Параметры рецептов Пластин
D00371	WORD	Параметры рецептов Пластин
D00372	WORD	Параметры рецептов Пластин
D00373	WORD	Параметры рецептов Пластин
D00374	WORD	Параметры рецептов Пластин
D00375	WORD	Параметры рецептов Пластин
D00376	WORD	Параметры рецептов Пластин
D00377	WORD	Параметры рецептов Пластин
D00378	WORD	Параметры рецептов Пластин
D00379	WORD	Параметры рецептов Пластин
D00380	WORD	Параметры рецептов Пластин
D00381	WORD	Параметры рецептов Пластин
D00382	WORD	Параметры рецептов Пластин
D00383	WORD	Параметры рецептов Пластин
D00384	WORD	Параметры рецептов Пластин
D00385	WORD	Параметры рецептов Пластин
D00386	WORD	Параметры рецептов Пластин
D00387	WORD	Параметры рецептов Пластин
D00388	WORD	Параметры рецептов Пластин
D00389	WORD	Параметры рецептов Пластин
D00390	WORD	Параметры рецептов Пластин
D00391	WORD	Параметры рецептов Пластин
D00392	WORD	Параметры рецептов Пластин
D00393	WORD	Параметры рецептов Пластин
D00394	WORD	Параметры рецептов Пластин
D00395	WORD	Параметры рецептов Пластин
D00396	WORD	Параметры рецептов Пластин
D00397	WORD	Параметры рецептов Пластин
D00398	WORD	Параметры рецептов Пластин
D00399	WORD	Параметры рецептов Пластин
D00408	WORD	Параметры рецептов заданий
D00409	WORD	Параметры рецептов заданий
D00410	WORD	Параметры рецептов заданий
D00411	WORD	Параметры рецептов заданий
D00412	WORD	Параметры рецептов заданий
D00413	WORD	Параметры рецептов заданий
D00414	WORD	Параметры рецептов заданий
D00415	WORD	Параметры рецептов заданий
D00416	WORD	Параметры рецептов заданий
D00417	WORD	Параметры рецептов заданий
D00418	WORD	Параметры рецептов заданий
D00419	WORD	Параметры рецептов заданий
D00420	WORD	Параметры рецептов заданий
D00421	WORD	Параметры рецептов заданий
D00422	WORD	Параметры рецептов заданий
D00423	WORD	Параметры рецептов заданий
D00424	WORD	Параметры рецептов заданий
D00425	WORD	Параметры рецептов заданий
D00426	WORD	Параметры рецептов заданий
D00427	WORD	Параметры рецептов заданий
D00428	WORD	Параметры рецептов заданий
D00429	WORD	Параметры рецептов заданий
D00430	WORD	Параметры рецептов заданий
D00431	WORD	Параметры рецептов заданий
D00432	WORD	Параметры рецептов заданий
D00433	WORD	Параметры рецептов заданий
D00434	WORD	Параметры рецептов заданий
D00435	WORD	Параметры рецептов заданий
D00436	WORD	Параметры рецептов заданий
D00437	WORD	Параметры рецептов заданий
D00438	WORD	Параметры рецептов заданий
D00439	WORD	Параметры рецептов заданий
D00440	WORD	Параметры рецептов заданий
D00441	WORD	Параметры рецептов заданий
D00442	WORD	Параметры рецептов заданий
D00443	WORD	Параметры рецептов заданий
D00444	WORD	Параметры рецептов заданий
D00445	WORD	Параметры рецептов заданий
D00446	WORD	Параметры рецептов заданий
D00447	WORD	Параметры рецептов заданий
D00448	WORD	Параметры рецептов заданий
D00449	WORD	Параметры рецептов заданий
D00450	WORD	Параметры рецептов заданий
D00451	WORD	Параметры рецептов заданий
D00452	WORD	Параметры рецептов заданий
D00453	WORD	Параметры рецептов заданий
D00454	WORD	Параметры рецептов заданий
D00455	WORD	Параметры рецептов заданий
D00456	WORD	Параметры рецептов заданий
D00457	WORD	Параметры рецептов заданий
D00458	WORD	Параметры рецептов заданий
D00459	WORD	Параметры рецептов заданий
D00460	WORD	Параметры рецептов заданий
D00461	WORD	Параметры рецептов заданий
D00462	WORD	Параметры рецептов заданий
D00463	WORD	Параметры рецептов заданий
D00464	WORD	Параметры рецептов заданий
D00465	WORD	Параметры рецептов заданий
D00466	WORD	Параметры рецептов заданий
D00467	WORD	Параметры рецептов заданий
D00468	WORD	Параметры рецептов заданий
D00469	WORD	Параметры рецептов заданий
D00470	WORD	Параметры рецептов заданий
D00471	WORD	Параметры рецептов заданий
D00472	WORD	Параметры рецептов заданий
D00473	WORD	Параметры рецептов заданий
D00474	WORD	Параметры рецептов заданий
D00475	WORD	Параметры рецептов заданий
D00476	WORD	Параметры рецептов заданий
D00477	WORD	Параметры рецептов заданий
D00478	WORD	Параметры рецептов заданий
D00479	WORD	Параметры рецептов заданий
D00480	WORD	Параметры рецептов заданий
D00481	WORD	Параметры рецептов заданий
D00482	WORD	Параметры рецептов заданий
D00483	WORD	Параметры рецептов заданий
D00484	WORD	Параметры рецептов заданий
D00485	WORD	Параметры рецептов заданий
D00486	WORD	Параметры рецептов заданий
D00487	WORD	Параметры рецептов заданий
D00488	WORD	Параметры рецептов заданий
D00489	WORD	Параметры рецептов заданий
D00490	WORD	Параметры рецептов заданий
D00491	WORD	Параметры рецептов заданий
D00492	WORD	Параметры рецептов заданий
D00493	WORD	Параметры рецептов заданий
D00494	WORD	Параметры рецептов заданий
D00495	WORD	Параметры рецептов заданий
D00496	WORD	Параметры рецептов заданий
D00497	WORD	Параметры рецептов заданий
D00498	WORD	Параметры рецептов заданий
D00499	WORD	Параметры рецептов заданий
D00143	WORD	MULNULL
D00144	WORD	MULNULL
D00145	WORD	MULNULL
D00148	WORD	MULNULL
D00149	WORD	MULNULL
D00150	WORD	MULNULL
D00152	WORD	MULNULL
D00153	WORD	MULNULL
D00154	WORD	MULNULL
D00159	WORD	MULNULL
D00160	WORD	MULNULL
D00161	WORD	MULNULL
D00163	WORD	MULNULL
D00164	WORD	MULNULL
D00165	WORD	MULNULL
D10001	WORD	Память для хранения названий рецептов. Задание 1. Символы 3-4
D10002	WORD	Память для хранения названий рецептов. Задание 1. Символы 5-6
D10003	WORD	Память для хранения названий рецептов. Задание 1. Символы 7-8
D10004	WORD	Память для хранения названий рецептов. Задание 1. Символы 9-10
D10005	WORD	Память для хранения названий рецептов. Задание 1. Символы 11-12
D10006	WORD	Память для хранения названий рецептов. Задание 1. Символы 13-14
D10007	WORD	Память для хранения названий рецептов. Задание 1. Символы 15-16
D10008	WORD	Память для хранения названий рецептов. Задание 1. Символы 17-18
D10009	WORD	Память для хранения названий рецептов. Задание 1. Символы 19-20
D10010	WORD	Память для хранения названий рецептов. Задание 1. Символы 21-22
D10011	WORD	Память для хранения названий рецептов. Задание 1. Символы 23-24
D10012	WORD	Память для хранения названий рецептов. Задание 1. Символы 25-26
D10013	WORD	Память для хранения названий рецептов. Задание 1. Символы 27-28
D10014	WORD	Память для хранения названий рецептов. Задание 1. Символы 29-30
D10015	WORD	Память для хранения названий рецептов. Задание 1. Символы 31-32
D10016	WORD	Память для хранения названий рецептов. Задание 2. Символы 1-2
D10017	WORD	Память для хранения названий рецептов. Задание 2. Символы 3-4
D10018	WORD	Память для хранения названий рецептов. Задание 2. Символы 5-6
D10019	WORD	Память для хранения названий рецептов. Задание 2. Символы 7-8
D10020	WORD	Память для хранения названий рецептов. Задание 2. Символы 9-10
D10021	WORD	Память для хранения названий рецептов. Задание 2. Символы 11-12
D10022	WORD	Память для хранения названий рецептов. Задание 2. Символы 13-14
D10023	WORD	Память для хранения названий рецептов. Задание 2. Символы 15-16
D10024	WORD	Память для хранения названий рецептов. Задание 2. Символы 17-18
D10025	WORD	Память для хранения названий рецептов. Задание 2. Символы 19-20
D10026	WORD	Память для хранения названий рецептов. Задание 2. Символы 21-22
D10027	WORD	Память для хранения названий рецептов. Задание 2. Символы 23-24
D10028	WORD	Память для хранения названий рецептов. Задание 2. Символы 25-26
D10029	WORD	Память для хранения названий рецептов. Задание 2. Символы 27-28
D10030	WORD	Память для хранения названий рецептов. Задание 2. Символы 29-30
D10031	WORD	Память для хранения названий рецептов. Задание 2. Символы 31-32
D10032	WORD	Память для хранения названий рецептов. Задание 3. Символы 1-2
D10033	WORD	Память для хранения названий рецептов. Задание 3. Символы 3-4
D10034	WORD	Память для хранения названий рецептов. Задание 3. Символы 5-6
D10035	WORD	Память для хранения названий рецептов. Задание 3. Символы 7-8
D10036	WORD	Память для хранения названий рецептов. Задание 3. Символы 9-10
D10037	WORD	Память для хранения названий рецептов. Задание 3. Символы 11-12
D10038	WORD	Память для хранения названий рецептов. Задание 3. Символы 13-14
D10039	WORD	Память для хранения названий рецептов. Задание 3. Символы 15-16
D10040	WORD	Память для хранения названий рецептов. Задание 3. Символы 17-18
D10041	WORD	Память для хранения названий рецептов. Задание 3. Символы 19-20
D10042	WORD	Память для хранения названий рецептов. Задание 3. Символы 21-22
D10043	WORD	Память для хранения названий рецептов. Задание 3. Символы 23-24
D10044	WORD	Память для хранения названий рецептов. Задание 3. Символы 25-26
D10045	WORD	Память для хранения названий рецептов. Задание 3. Символы 27-28
D10046	WORD	Память для хранения названий рецептов. Задание 3. Символы 29-30
D10047	WORD	Память для хранения названий рецептов. Задание 3. Символы 31-32
D10048	WORD	Память для хранения названий рецептов. Задание 4. Символы 1-2
D10049	WORD	Память для хранения названий рецептов. Задание 4. Символы 3-4
D10050	WORD	Память для хранения названий рецептов. Задание 4. Символы 5-6
D10051	WORD	Память для хранения названий рецептов. Задание 4. Символы 7-8
D10052	WORD	Память для хранения названий рецептов. Задание 4. Символы 9-10
D10053	WORD	Память для хранения названий рецептов. Задание 4. Символы 11-12
D10054	WORD	Память для хранения названий рецептов. Задание 4. Символы 13-14
D10055	WORD	Память для хранения названий рецептов. Задание 4. Символы 15-16
D10056	WORD	Память для хранения названий рецептов. Задание 4. Символы 17-18
D10057	WORD	Память для хранения названий рецептов. Задание 4. Символы 19-20
D10058	WORD	Память для хранения названий рецептов. Задание 4. Символы 21-22
D10059	WORD	Память для хранения названий рецептов. Задание 4. Символы 23-24
D10060	WORD	Память для хранения названий рецептов. Задание 4. Символы 25-26
D10061	WORD	Память для хранения названий рецептов. Задание 4. Символы 27-28
D10062	WORD	Память для хранения названий рецептов. Задание 4. Символы 29-30
D10063	WORD	Память для хранения названий рецептов. Задание 4. Символы 31-32
D10064	WORD	Память для хранения названий рецептов. Задание 5. Символы 1-2
D10065	WORD	Память для хранения названий рецептов. Задание 5. Символы 3-4
D10066	WORD	Память для хранения названий рецептов. Задание 5. Символы 5-6
D10067	WORD	Память для хранения названий рецептов. Задание 5. Символы 7-8
D10068	WORD	Память для хранения названий рецептов. Задание 5. Символы 9-10
D10069	WORD	Память для хранения названий рецептов. Задание 5. Символы 11-12
D10070	WORD	Память для хранения названий рецептов. Задание 5. Символы 13-14
D10071	WORD	Память для хранения названий рецептов. Задание 5. Символы 15-16
D10072	WORD	Память для хранения названий рецептов. Задание 5. Символы 17-18
D10073	WORD	Память для хранения названий рецептов. Задание 5. Символы 19-20
D10074	WORD	Память для хранения названий рецептов. Задание 5. Символы 21-22
D10075	WORD	Память для хранения названий рецептов. Задание 5. Символы 23-24
D10076	WORD	Память для хранения названий рецептов. Задание 5. Символы 25-26
D10077	WORD	Память для хранения названий рецептов. Задание 5. Символы 27-28
D10078	WORD	Память для хранения названий рецептов. Задание 5. Символы 29-30
D10079	WORD	Память для хранения названий рецептов. Задание 5. Символы 31-32
D10080	WORD	Память для хранения названий рецептов. Задание 6. Символы 1-2
D10081	WORD	Память для хранения названий рецептов. Задание 6. Символы 3-4
D10082	WORD	Память для хранения названий рецептов. Задание 6. Символы 5-6
D10083	WORD	Память для хранения названий рецептов. Задание 6. Символы 7-8
D10084	WORD	Память для хранения названий рецептов. Задание 6. Символы 9-10
D10085	WORD	Память для хранения названий рецептов. Задание 6. Символы 11-12
D10086	WORD	Память для хранения названий рецептов. Задание 6. Символы 13-14
D10087	WORD	Память для хранения названий рецептов. Задание 6. Символы 15-16
D10088	WORD	Память для хранения названий рецептов. Задание 6. Символы 17-18
D10089	WORD	Память для хранения названий рецептов. Задание 6. Символы 19-20
D10090	WORD	Память для хранения названий рецептов. Задание 6. Символы 21-22
D10091	WORD	Память для хранения названий рецептов. Задание 6. Символы 23-24
D10092	WORD	Память для хранения названий рецептов. Задание 6. Символы 25-26
D10093	WORD	Память для хранения названий рецептов. Задание 6. Символы 27-28
D10094	WORD	Память для хранения названий рецептов. Задание 6. Символы 29-30
D10095	WORD	Память для хранения названий рецептов. Задание 6. Символы 31-32
D10096	WORD	Память для хранения названий рецептов. Задание 7. Символы 1-2
D10097	WORD	Память для хранения названий рецептов. Задание 7. Символы 3-4
D10098	WORD	Память для хранения названий рецептов. Задание 7. Символы 5-6
D10099	WORD	Память для хранения названий рецептов. Задание 7. Символы 7-8
D10100	WORD	Память для хранения названий рецептов. Задание 7. Символы 9-10
D10101	WORD	Память для хранения названий рецептов. Задание 7. Символы 11-12
D10102	WORD	Память для хранения названий рецептов. Задание 7. Символы 13-14
D10103	WORD	Память для хранения названий рецептов. Задание 7. Символы 15-16
D10104	WORD	Память для хранения названий рецептов. Задание 7. Символы 17-18
D10105	WORD	Память для хранения названий рецептов. Задание 7. Символы 19-20
D10106	WORD	Память для хранения названий рецептов. Задание 7. Символы 21-22
D10107	WORD	Память для хранения названий рецептов. Задание 7. Символы 23-24
D10108	WORD	Память для хранения названий рецептов. Задание 7. Символы 25-26
D10109	WORD	Память для хранения названий рецептов. Задание 7. Символы 27-28
D10110	WORD	Память для хранения названий рецептов. Задание 7. Символы 29-30
D10111	WORD	Память для хранения названий рецептов. Задание 7. Символы 31-32
D10112	WORD	Память для хранения названий рецептов. Задание 8. Символы 1-2
D10113	WORD	Память для хранения названий рецептов. Задание 8. Символы 3-4
D10114	WORD	Память для хранения названий рецептов. Задание 8. Символы 5-6
D10115	WORD	Память для хранения названий рецептов. Задание 8. Символы 7-8
D10116	WORD	Память для хранения названий рецептов. Задание 8. Символы 9-10
D10117	WORD	Память для хранения названий рецептов. Задание 8. Символы 11-12
D10118	WORD	Память для хранения названий рецептов. Задание 8. Символы 13-14
D10119	WORD	Память для хранения названий рецептов. Задание 8. Символы 15-16
D10120	WORD	Память для хранения названий рецептов. Задание 8. Символы 17-18
D10121	WORD	Память для хранения названий рецептов. Задание 8. Символы 19-20
D10122	WORD	Память для хранения названий рецептов. Задание 8. Символы 21-22
D10123	WORD	Память для хранения названий рецептов. Задание 8. Символы 23-24
D10124	WORD	Память для хранения названий рецептов. Задание 8. Символы 25-26
D10125	WORD	Память для хранения названий рецептов. Задание 8. Символы 27-28
D10126	WORD	Память для хранения названий рецептов. Задание 8. Символы 29-30
D10127	WORD	Память для хранения названий рецептов. Задание 8. Символы 31-32
D10128	WORD	Память для хранения названий рецептов. Задание 9. Символы 1-2
D10129	WORD	Память для хранения названий рецептов. Задание 9. Символы 3-4
D10130	WORD	Память для хранения названий рецептов. Задание 9. Символы 5-6
D10131	WORD	Память для хранения названий рецептов. Задание 9. Символы 7-8
D10132	WORD	Память для хранения названий рецептов. Задание 9. Символы 9-10
D10133	WORD	Память для хранения названий рецептов. Задание 9. Символы 11-12
D10134	WORD	Память для хранения названий рецептов. Задание 9. Символы 13-14
D10135	WORD	Память для хранения названий рецептов. Задание 9. Символы 15-16
D10136	WORD	Память для хранения названий рецептов. Задание 9. Символы 17-18
D10137	WORD	Память для хранения названий рецептов. Задание 9. Символы 19-20
D10138	WORD	Память для хранения названий рецептов. Задание 9. Символы 21-22
D10139	WORD	Память для хранения названий рецептов. Задание 9. Символы 23-24
D10140	WORD	Память для хранения названий рецептов. Задание 9. Символы 25-26
D10141	WORD	Память для хранения названий рецептов. Задание 9. Символы 27-28
D10142	WORD	Память для хранения названий рецептов. Задание 9. Символы 29-30
D10143	WORD	Память для хранения названий рецептов. Задание 9. Символы 31-32
D10144	WORD	Память для хранения названий рецептов. Задание 10. Символы 1-2
D10145	WORD	Память для хранения названий рецептов. Задание 10. Символы 3-4
D10146	WORD	Память для хранения названий рецептов. Задание 10. Символы 5-6
D10147	WORD	Память для хранения названий рецептов. Задание 10. Символы 7-8
D10148	WORD	Память для хранения названий рецептов. Задание 10. Символы 9-10
D10149	WORD	Память для хранения названий рецептов. Задание 10. Символы 11-12
D10150	WORD	Память для хранения названий рецептов. Задание 10. Символы 13-14
D10151	WORD	Память для хранения названий рецептов. Задание 10. Символы 15-16
D10152	WORD	Память для хранения названий рецептов. Задание 10. Символы 17-18
D10153	WORD	Память для хранения названий рецептов. Задание 10. Символы 19-20
D10154	WORD	Память для хранения названий рецептов. Задание 10. Символы 21-22
D10155	WORD	Память для хранения названий рецептов. Задание 10. Символы 23-24
D10156	WORD	Память для хранения названий рецептов. Задание 10. Символы 25-26
D10157	WORD	Память для хранения названий рецептов. Задание 10. Символы 27-28
D10158	WORD	Память для хранения названий рецептов. Задание 10. Символы 29-30
D10159	WORD	Память для хранения названий рецептов. Задание 10. Символы 31-32
D10160	WORD	Память для хранения названий рецептов. Задание 11. Символы 1-2
D10161	WORD	Память для хранения названий рецептов. Задание 11. Символы 3-4
D10162	WORD	Память для хранения названий рецептов. Задание 11. Символы 5-6
D10163	WORD	Память для хранения названий рецептов. Задание 11. Символы 7-8
D10164	WORD	Память для хранения названий рецептов. Задание 11. Символы 9-10
D10165	WORD	Память для хранения названий рецептов. Задание 11. Символы 11-12
D10166	WORD	Память для хранения названий рецептов. Задание 11. Символы 13-14
D10167	WORD	Память для хранения названий рецептов. Задание 11. Символы 15-16
D10168	WORD	Память для хранения названий рецептов. Задание 11. Символы 17-18
D10169	WORD	Память для хранения названий рецептов. Задание 11. Символы 19-20
D10170	WORD	Память для хранения названий рецептов. Задание 11. Символы 21-22
D10171	WORD	Память для хранения названий рецептов. Задание 11. Символы 23-24
D10172	WORD	Память для хранения названий рецептов. Задание 11. Символы 25-26
D10173	WORD	Память для хранения названий рецептов. Задание 11. Символы 27-28
D10174	WORD	Память для хранения названий рецептов. Задание 11. Символы 29-30
D10175	WORD	Память для хранения названий рецептов. Задание 11. Символы 31-32
D10176	WORD	Память для хранения названий рецептов. Задание 12. Символы 1-2
D10177	WORD	Память для хранения названий рецептов. Задание 12. Символы 3-4
D10178	WORD	Память для хранения названий рецептов. Задание 12. Символы 5-6
D10179	WORD	Память для хранения названий рецептов. Задание 12. Символы 7-8
D10180	WORD	Память для хранения названий рецептов. Задание 12. Символы 9-10
D10181	WORD	Память для хранения названий рецептов. Задание 12. Символы 11-12
D10182	WORD	Память для хранения названий рецептов. Задание 12. Символы 13-14
D10183	WORD	Память для хранения названий рецептов. Задание 12. Символы 15-16
D10184	WORD	Память для хранения названий рецептов. Задание 12. Символы 17-18
D10185	WORD	Память для хранения названий рецептов. Задание 12. Символы 19-20
D10186	WORD	Память для хранения названий рецептов. Задание 12. Символы 21-22
D10187	WORD	Память для хранения названий рецептов. Задание 12. Символы 23-24
D10188	WORD	Память для хранения названий рецептов. Задание 12. Символы 25-26
D10189	WORD	Память для хранения названий рецептов. Задание 12. Символы 27-28
D10190	WORD	Память для хранения названий рецептов. Задание 12. Символы 29-30
D10191	WORD	Память для хранения названий рецептов. Задание 12. Символы 31-32
D10192	WORD	Память для хранения названий рецептов. Задание 13. Символы 1-2
D10193	WORD	Память для хранения названий рецептов. Задание 13. Символы 3-4
D10194	WORD	Память для хранения названий рецептов. Задание 13. Символы 5-6
D10195	WORD	Память для хранения названий рецептов. Задание 13. Символы 7-8
D10196	WORD	Память для хранения названий рецептов. Задание 13. Символы 9-10
D10197	WORD	Память для хранения названий рецептов. Задание 13. Символы 11-12
D10198	WORD	Память для хранения названий рецептов. Задание 13. Символы 13-14
D10199	WORD	Память для хранения названий рецептов. Задание 13. Символы 15-16
D10200	WORD	Память для хранения названий рецептов. Задание 13. Символы 17-18
D10201	WORD	Память для хранения названий рецептов. Задание 13. Символы 19-20
D10202	WORD	Память для хранения названий рецептов. Задание 13. Символы 21-22
D10203	WORD	Память для хранения названий рецептов. Задание 13. Символы 23-24
D10204	WORD	Память для хранения названий рецептов. Задание 13. Символы 25-26
D10205	WORD	Память для хранения названий рецептов. Задание 13. Символы 27-28
D10206	WORD	Память для хранения названий рецептов. Задание 13. Символы 29-30
D10207	WORD	Память для хранения названий рецептов. Задание 13. Символы 31-32
D10208	WORD	Память для хранения названий рецептов. Задание 14. Символы 1-2
D10209	WORD	Память для хранения названий рецептов. Задание 14. Символы 3-4
D10210	WORD	Память для хранения названий рецептов. Задание 14. Символы 5-6
D10211	WORD	Память для хранения названий рецептов. Задание 14. Символы 7-8
D10212	WORD	Память для хранения названий рецептов. Задание 14. Символы 9-10
D10213	WORD	Память для хранения названий рецептов. Задание 14. Символы 11-12
D10214	WORD	Память для хранения названий рецептов. Задание 14. Символы 13-14
D10215	WORD	Память для хранения названий рецептов. Задание 14. Символы 15-16
D10216	WORD	Память для хранения названий рецептов. Задание 14. Символы 17-18
D10217	WORD	Память для хранения названий рецептов. Задание 14. Символы 19-20
D10218	WORD	Память для хранения названий рецептов. Задание 14. Символы 21-22
D10219	WORD	Память для хранения названий рецептов. Задание 14. Символы 23-24
D10220	WORD	Память для хранения названий рецептов. Задание 14. Символы 25-26
D10221	WORD	Память для хранения названий рецептов. Задание 14. Символы 27-28
D10222	WORD	Память для хранения названий рецептов. Задание 14. Символы 29-30
D10223	WORD	Память для хранения названий рецептов. Задание 14. Символы 31-32
D10224	WORD	Память для хранения названий рецептов. Задание 15. Символы 1-2
D10225	WORD	Память для хранения названий рецептов. Задание 15. Символы 3-4
D10226	WORD	Память для хранения названий рецептов. Задание 15. Символы 5-6
D10227	WORD	Память для хранения названий рецептов. Задание 15. Символы 7-8
D10228	WORD	Память для хранения названий рецептов. Задание 15. Символы 9-10
D10229	WORD	Память для хранения названий рецептов. Задание 15. Символы 11-12
D10230	WORD	Память для хранения названий рецептов. Задание 15. Символы 13-14
D10231	WORD	Память для хранения названий рецептов. Задание 15. Символы 15-16
D10232	WORD	Память для хранения названий рецептов. Задание 15. Символы 17-18
D10233	WORD	Память для хранения названий рецептов. Задание 15. Символы 19-20
D10234	WORD	Память для хранения названий рецептов. Задание 15. Символы 21-22
D10235	WORD	Память для хранения названий рецептов. Задание 15. Символы 23-24
D10236	WORD	Память для хранения названий рецептов. Задание 15. Символы 25-26
D10237	WORD	Память для хранения названий рецептов. Задание 15. Символы 27-28
D10238	WORD	Память для хранения названий рецептов. Задание 15. Символы 29-30
D10239	WORD	Память для хранения названий рецептов. Задание 15. Символы 31-32
D10240	WORD	Память для хранения названий рецептов. Задание 16. Символы 1-2
D10241	WORD	Память для хранения названий рецептов. Задание 16. Символы 3-4
D10242	WORD	Память для хранения названий рецептов. Задание 16. Символы 5-6
D10243	WORD	Память для хранения названий рецептов. Задание 16. Символы 7-8
D10244	WORD	Память для хранения названий рецептов. Задание 16. Символы 9-10
D10245	WORD	Память для хранения названий рецептов. Задание 16. Символы 11-12
D10246	WORD	Память для хранения названий рецептов. Задание 16. Символы 13-14
D10247	WORD	Память для хранения названий рецептов. Задание 16. Символы 15-16
D10248	WORD	Память для хранения названий рецептов. Задание 16. Символы 17-18
D10249	WORD	Память для хранения названий рецептов. Задание 16. Символы 19-20
D10250	WORD	Память для хранения названий рецептов. Задание 16. Символы 21-22
D10251	WORD	Память для хранения названий рецептов. Задание 16. Символы 23-24
D10252	WORD	Память для хранения названий рецептов. Задание 16. Символы 25-26
D10253	WORD	Память для хранения названий рецептов. Задание 16. Символы 27-28
D10254	WORD	Память для хранения названий рецептов. Задание 16. Символы 29-30
D10255	WORD	Память для хранения названий рецептов. Задание 16. Символы 31-32
D10256	WORD	Память для хранения названий рецептов. Задание 17. Символы 1-2
D10257	WORD	Память для хранения названий рецептов. Задание 17. Символы 3-4
D10258	WORD	Память для хранения названий рецептов. Задание 17. Символы 5-6
D10259	WORD	Память для хранения названий рецептов. Задание 17. Символы 7-8
D10260	WORD	Память для хранения названий рецептов. Задание 17. Символы 9-10
D10261	WORD	Память для хранения названий рецептов. Задание 17. Символы 11-12
D10262	WORD	Память для хранения названий рецептов. Задание 17. Символы 13-14
D10263	WORD	Память для хранения названий рецептов. Задание 17. Символы 15-16
D10264	WORD	Память для хранения названий рецептов. Задание 17. Символы 17-18
D10265	WORD	Память для хранения названий рецептов. Задание 17. Символы 19-20
D10266	WORD	Память для хранения названий рецептов. Задание 17. Символы 21-22
D10267	WORD	Память для хранения названий рецептов. Задание 17. Символы 23-24
D10268	WORD	Память для хранения названий рецептов. Задание 17. Символы 25-26
D10269	WORD	Память для хранения названий рецептов. Задание 17. Символы 27-28
D10270	WORD	Память для хранения названий рецептов. Задание 17. Символы 29-30
D10271	WORD	Память для хранения названий рецептов. Задание 17. Символы 31-32
D10272	WORD	Память для хранения названий рецептов. Задание 18. Символы 1-2
D10273	WORD	Память для хранения названий рецептов. Задание 18. Символы 3-4
D10274	WORD	Память для хранения названий рецептов. Задание 18. Символы 5-6
D10275	WORD	Память для хранения названий рецептов. Задание 18. Символы 7-8
D10276	WORD	Память для хранения названий рецептов. Задание 18. Символы 9-10
D10277	WORD	Память для хранения названий рецептов. Задание 18. Символы 11-12
D10278	WORD	Память для хранения названий рецептов. Задание 18. Символы 13-14
D10279	WORD	Память для хранения названий рецептов. Задание 18. Символы 15-16
D10280	WORD	Память для хранения названий рецептов. Задание 18. Символы 17-18
D10281	WORD	Память для хранения названий рецептов. Задание 18. Символы 19-20
D10282	WORD	Память для хранения названий рецептов. Задание 18. Символы 21-22
D10283	WORD	Память для хранения названий рецептов. Задание 18. Символы 23-24
D10284	WORD	Память для хранения названий рецептов. Задание 18. Символы 25-26
D10285	WORD	Память для хранения названий рецептов. Задание 18. Символы 27-28
D10286	WORD	Память для хранения названий рецептов. Задание 18. Символы 29-30
D10287	WORD	Память для хранения названий рецептов. Задание 18. Символы 31-32
D10288	WORD	Память для хранения названий рецептов. Задание 19. Символы 1-2
D10289	WORD	Память для хранения названий рецептов. Задание 19. Символы 3-4
D10290	WORD	Память для хранения названий рецептов. Задание 19. Символы 5-6
D10291	WORD	Память для хранения названий рецептов. Задание 19. Символы 7-8
D10292	WORD	Память для хранения названий рецептов. Задание 19. Символы 9-10
D10293	WORD	Память для хранения названий рецептов. Задание 19. Символы 11-12
D10294	WORD	Память для хранения названий рецептов. Задание 19. Символы 13-14
D10295	WORD	Память для хранения названий рецептов. Задание 19. Символы 15-16
D10296	WORD	Память для хранения названий рецептов. Задание 19. Символы 17-18
D10297	WORD	Память для хранения названий рецептов. Задание 19. Символы 19-20
D10298	WORD	Память для хранения названий рецептов. Задание 19. Символы 21-22
D10299	WORD	Память для хранения названий рецептов. Задание 19. Символы 23-24
D10300	WORD	Память для хранения названий рецептов. Задание 19. Символы 25-26
D10301	WORD	Память для хранения названий рецептов. Задание 19. Символы 27-28
D10302	WORD	Память для хранения названий рецептов. Задание 19. Символы 29-30
D10303	WORD	Память для хранения названий рецептов. Задание 19. Символы 31-32
D10304	WORD	Память для хранения названий рецептов. Задание 20. Символы 1-2
D10305	WORD	Память для хранения названий рецептов. Задание 20. Символы 3-4
D10306	WORD	Память для хранения названий рецептов. Задание 20. Символы 5-6
D10307	WORD	Память для хранения названий рецептов. Задание 20. Символы 7-8
D10308	WORD	Память для хранения названий рецептов. Задание 20. Символы 9-10
D10309	WORD	Память для хранения названий рецептов. Задание 20. Символы 11-12
D10310	WORD	Память для хранения названий рецептов. Задание 20. Символы 13-14
D10311	WORD	Память для хранения названий рецептов. Задание 20. Символы 15-16
D10312	WORD	Память для хранения названий рецептов. Задание 20. Символы 17-18
D10313	WORD	Память для хранения названий рецептов. Задание 20. Символы 19-20
D10314	WORD	Память для хранения названий рецептов. Задание 20. Символы 21-22
D10315	WORD	Память для хранения названий рецептов. Задание 20. Символы 23-24
D10316	WORD	Память для хранения названий рецептов. Задание 20. Символы 25-26
D10317	WORD	Память для хранения названий рецептов. Задание 20. Символы 27-28
D10318	WORD	Память для хранения названий рецептов. Задание 20. Символы 29-30
D10319	WORD	Память для хранения названий рецептов. Задание 20. Символы 31-32
D10320	WORD	Память для хранения названий рецептов. Задание 21. Символы 1-2
D10321	WORD	Память для хранения названий рецептов. Задание 21. Символы 3-4
D10322	WORD	Память для хранения названий рецептов. Задание 21. Символы 5-6
D10323	WORD	Память для хранения названий рецептов. Задание 21. Символы 7-8
D10324	WORD	Память для хранения названий рецептов. Задание 21. Символы 9-10
D10325	WORD	Память для хранения названий рецептов. Задание 21. Символы 11-12
D10326	WORD	Память для хранения названий рецептов. Задание 21. Символы 13-14
D10327	WORD	Память для хранения названий рецептов. Задание 21. Символы 15-16
D10328	WORD	Память для хранения названий рецептов. Задание 21. Символы 17-18
D10329	WORD	Память для хранения названий рецептов. Задание 21. Символы 19-20
D10330	WORD	Память для хранения названий рецептов. Задание 21. Символы 21-22
D10331	WORD	Память для хранения названий рецептов. Задание 21. Символы 23-24
D10332	WORD	Память для хранения названий рецептов. Задание 21. Символы 25-26
D10333	WORD	Память для хранения названий рецептов. Задание 21. Символы 27-28
D10334	WORD	Память для хранения названий рецептов. Задание 21. Символы 29-30
D10335	WORD	Память для хранения названий рецептов. Задание 21. Символы 31-32
D10336	WORD	Память для хранения названий рецептов. Задание 22. Символы 1-2
D10337	WORD	Память для хранения названий рецептов. Задание 22. Символы 3-4
D10338	WORD	Память для хранения названий рецептов. Задание 22. Символы 5-6
D10339	WORD	Память для хранения названий рецептов. Задание 22. Символы 7-8
D10340	WORD	Память для хранения названий рецептов. Задание 22. Символы 9-10
D10341	WORD	Память для хранения названий рецептов. Задание 22. Символы 11-12
D10342	WORD	Память для хранения названий рецептов. Задание 22. Символы 13-14
D10343	WORD	Память для хранения названий рецептов. Задание 22. Символы 15-16
D10344	WORD	Память для хранения названий рецептов. Задание 22. Символы 17-18
D10345	WORD	Память для хранения названий рецептов. Задание 22. Символы 19-20
D10346	WORD	Память для хранения названий рецептов. Задание 22. Символы 21-22
D10347	WORD	Память для хранения названий рецептов. Задание 22. Символы 23-24
D10348	WORD	Память для хранения названий рецептов. Задание 22. Символы 25-26
D10349	WORD	Память для хранения названий рецептов. Задание 22. Символы 27-28
D10350	WORD	Память для хранения названий рецептов. Задание 22. Символы 29-30
D10351	WORD	Память для хранения названий рецептов. Задание 22. Символы 31-32
D10352	WORD	Память для хранения названий рецептов. Задание 23. Символы 1-2
D10353	WORD	Память для хранения названий рецептов. Задание 23. Символы 3-4
D10354	WORD	Память для хранения названий рецептов. Задание 23. Символы 5-6
D10355	WORD	Память для хранения названий рецептов. Задание 23. Символы 7-8
D10356	WORD	Память для хранения названий рецептов. Задание 23. Символы 9-10
D10357	WORD	Память для хранения названий рецептов. Задание 23. Символы 11-12
D10358	WORD	Память для хранения названий рецептов. Задание 23. Символы 13-14
D10359	WORD	Память для хранения названий рецептов. Задание 23. Символы 15-16
D10360	WORD	Память для хранения названий рецептов. Задание 23. Символы 17-18
D10361	WORD	Память для хранения названий рецептов. Задание 23. Символы 19-20
D10362	WORD	Память для хранения названий рецептов. Задание 23. Символы 21-22
D10363	WORD	Память для хранения названий рецептов. Задание 23. Символы 23-24
D10364	WORD	Память для хранения названий рецептов. Задание 23. Символы 25-26
D10365	WORD	Память для хранения названий рецептов. Задание 23. Символы 27-28
D10366	WORD	Память для хранения названий рецептов. Задание 23. Символы 29-30
D10367	WORD	Память для хранения названий рецептов. Задание 23. Символы 31-32
D10368	WORD	Память для хранения названий рецептов. Задание 24. Символы 1-2
D10369	WORD	Память для хранения названий рецептов. Задание 24. Символы 3-4
D10370	WORD	Память для хранения названий рецептов. Задание 24. Символы 5-6
D10371	WORD	Память для хранения названий рецептов. Задание 24. Символы 7-8
D10372	WORD	Память для хранения названий рецептов. Задание 24. Символы 9-10
D10373	WORD	Память для хранения названий рецептов. Задание 24. Символы 11-12
D10374	WORD	Память для хранения названий рецептов. Задание 24. Символы 13-14
D10375	WORD	Память для хранения названий рецептов. Задание 24. Символы 15-16
D10376	WORD	Память для хранения названий рецептов. Задание 24. Символы 17-18
D10377	WORD	Память для хранения названий рецептов. Задание 24. Символы 19-20
D10378	WORD	Память для хранения названий рецептов. Задание 24. Символы 21-22
D10379	WORD	Память для хранения названий рецептов. Задание 24. Символы 23-24
D10380	WORD	Память для хранения названий рецептов. Задание 24. Символы 25-26
D10381	WORD	Память для хранения названий рецептов. Задание 24. Символы 27-28
D10382	WORD	Память для хранения названий рецептов. Задание 24. Символы 29-30
D10383	WORD	Память для хранения названий рецептов. Задание 24. Символы 31-32
D10384	WORD	Память для хранения названий рецептов. Задание 25. Символы 1-2
D10385	WORD	Память для хранения названий рецептов. Задание 25. Символы 3-4
D10386	WORD	Память для хранения названий рецептов. Задание 25. Символы 5-6
D10387	WORD	Память для хранения названий рецептов. Задание 25. Символы 7-8
D10388	WORD	Память для хранения названий рецептов. Задание 25. Символы 9-10
D10389	WORD	Память для хранения названий рецептов. Задание 25. Символы 11-12
D10390	WORD	Память для хранения названий рецептов. Задание 25. Символы 13-14
D10391	WORD	Память для хранения названий рецептов. Задание 25. Символы 15-16
D10392	WORD	Память для хранения названий рецептов. Задание 25. Символы 17-18
D10393	WORD	Память для хранения названий рецептов. Задание 25. Символы 19-20
D10394	WORD	Память для хранения названий рецептов. Задание 25. Символы 21-22
D10395	WORD	Память для хранения названий рецептов. Задание 25. Символы 23-24
D10396	WORD	Память для хранения названий рецептов. Задание 25. Символы 25-26
D10397	WORD	Память для хранения названий рецептов. Задание 25. Символы 27-28
D10398	WORD	Память для хранения названий рецептов. Задание 25. Символы 29-30
D10399	WORD	Память для хранения названий рецептов. Задание 25. Символы 31-32
D10400	WORD	Память для хранения названий рецептов. Задание 26. Символы 1-2
D10401	WORD	Память для хранения названий рецептов. Задание 26. Символы 3-4
D10402	WORD	Память для хранения названий рецептов. Задание 26. Символы 5-6
D10403	WORD	Память для хранения названий рецептов. Задание 26. Символы 7-8
D10404	WORD	Память для хранения названий рецептов. Задание 26. Символы 9-10
D10405	WORD	Память для хранения названий рецептов. Задание 26. Символы 11-12
D10406	WORD	Память для хранения названий рецептов. Задание 26. Символы 13-14
D10407	WORD	Память для хранения названий рецептов. Задание 26. Символы 15-16
D10408	WORD	Память для хранения названий рецептов. Задание 26. Символы 17-18
D10409	WORD	Память для хранения названий рецептов. Задание 26. Символы 19-20
D10410	WORD	Память для хранения названий рецептов. Задание 26. Символы 21-22
D10411	WORD	Память для хранения названий рецептов. Задание 26. Символы 23-24
D10412	WORD	Память для хранения названий рецептов. Задание 26. Символы 25-26
D10413	WORD	Память для хранения названий рецептов. Задание 26. Символы 27-28
D10414	WORD	Память для хранения названий рецептов. Задание 26. Символы 29-30
D10415	WORD	Память для хранения названий рецептов. Задание 26. Символы 31-32
D10416	WORD	Память для хранения названий рецептов. Задание 27. Символы 1-2
D10417	WORD	Память для хранения названий рецептов. Задание 27. Символы 3-4
D10418	WORD	Память для хранения названий рецептов. Задание 27. Символы 5-6
D10419	WORD	Память для хранения названий рецептов. Задание 27. Символы 7-8
D10420	WORD	Память для хранения названий рецептов. Задание 27. Символы 9-10
D10421	WORD	Память для хранения названий рецептов. Задание 27. Символы 11-12
D10422	WORD	Память для хранения названий рецептов. Задание 27. Символы 13-14
D10423	WORD	Память для хранения названий рецептов. Задание 27. Символы 15-16
D10424	WORD	Память для хранения названий рецептов. Задание 27. Символы 17-18
D10425	WORD	Память для хранения названий рецептов. Задание 27. Символы 19-20
D10426	WORD	Память для хранения названий рецептов. Задание 27. Символы 21-22
D10427	WORD	Память для хранения названий рецептов. Задание 27. Символы 23-24
D10428	WORD	Память для хранения названий рецептов. Задание 27. Символы 25-26
D10429	WORD	Память для хранения названий рецептов. Задание 27. Символы 27-28
D10430	WORD	Память для хранения названий рецептов. Задание 27. Символы 29-30
D10431	WORD	Память для хранения названий рецептов. Задание 27. Символы 31-32
D10432	WORD	Память для хранения названий рецептов. Задание 28. Символы 1-2
D10433	WORD	Память для хранения названий рецептов. Задание 28. Символы 3-4
D10434	WORD	Память для хранения названий рецептов. Задание 28. Символы 5-6
D10435	WORD	Память для хранения названий рецептов. Задание 28. Символы 7-8
D10436	WORD	Память для хранения названий рецептов. Задание 28. Символы 9-10
D10437	WORD	Память для хранения названий рецептов. Задание 28. Символы 11-12
D10438	WORD	Память для хранения названий рецептов. Задание 28. Символы 13-14
D10439	WORD	Память для хранения названий рецептов. Задание 28. Символы 15-16
D10440	WORD	Память для хранения названий рецептов. Задание 28. Символы 17-18
D10441	WORD	Память для хранения названий рецептов. Задание 28. Символы 19-20
D10442	WORD	Память для хранения названий рецептов. Задание 28. Символы 21-22
D10443	WORD	Память для хранения названий рецептов. Задание 28. Символы 23-24
D10444	WORD	Память для хранения названий рецептов. Задание 28. Символы 25-26
D10445	WORD	Память для хранения названий рецептов. Задание 28. Символы 27-28
D10446	WORD	Память для хранения названий рецептов. Задание 28. Символы 29-30
D10447	WORD	Память для хранения названий рецептов. Задание 28. Символы 31-32
D10448	WORD	Память для хранения названий рецептов. Задание 29. Символы 1-2
D10449	WORD	Память для хранения названий рецептов. Задание 29. Символы 3-4
D10450	WORD	Память для хранения названий рецептов. Задание 29. Символы 5-6
D10451	WORD	Память для хранения названий рецептов. Задание 29. Символы 7-8
D10452	WORD	Память для хранения названий рецептов. Задание 29. Символы 9-10
D10453	WORD	Память для хранения названий рецептов. Задание 29. Символы 11-12
D10454	WORD	Память для хранения названий рецептов. Задание 29. Символы 13-14
D10455	WORD	Память для хранения названий рецептов. Задание 29. Символы 15-16
D10456	WORD	Память для хранения названий рецептов. Задание 29. Символы 17-18
D10457	WORD	Память для хранения названий рецептов. Задание 29. Символы 19-20
D10458	WORD	Память для хранения названий рецептов. Задание 29. Символы 21-22
D10459	WORD	Память для хранения названий рецептов. Задание 29. Символы 23-24
D10460	WORD	Память для хранения названий рецептов. Задание 29. Символы 25-26
D10461	WORD	Память для хранения названий рецептов. Задание 29. Символы 27-28
D10462	WORD	Память для хранения названий рецептов. Задание 29. Символы 29-30
D10463	WORD	Память для хранения названий рецептов. Задание 29. Символы 31-32
D10464	WORD	Память для хранения названий рецептов. Задание 30. Символы 1-2
D10465	WORD	Память для хранения названий рецептов. Задание 30. Символы 3-4
D10466	WORD	Память для хранения названий рецептов. Задание 30. Символы 5-6
D10467	WORD	Память для хранения названий рецептов. Задание 30. Символы 7-8
D10468	WORD	Память для хранения названий рецептов. Задание 30. Символы 9-10
D10469	WORD	Память для хранения названий рецептов. Задание 30. Символы 11-12
D10470	WORD	Память для хранения названий рецептов. Задание 30. Символы 13-14
D10471	WORD	Память для хранения названий рецептов. Задание 30. Символы 15-16
D10472	WORD	Память для хранения названий рецептов. Задание 30. Символы 17-18
D10473	WORD	Память для хранения названий рецептов. Задание 30. Символы 19-20
D10474	WORD	Память для хранения названий рецептов. Задание 30. Символы 21-22
D10475	WORD	Память для хранения названий рецептов. Задание 30. Символы 23-24
D10476	WORD	Память для хранения названий рецептов. Задание 30. Символы 25-26
D10477	WORD	Память для хранения названий рецептов. Задание 30. Символы 27-28
D10478	WORD	Память для хранения названий рецептов. Задание 30. Символы 29-30
D10479	WORD	Память для хранения названий рецептов. Задание 30. Символы 31-32
D10480	WORD	Память для хранения названий рецептов. Задание 31. Символы 1-2
D10481	WORD	Память для хранения названий рецептов. Задание 31. Символы 3-4
D10482	WORD	Память для хранения названий рецептов. Задание 31. Символы 5-6
D10483	WORD	Память для хранения названий рецептов. Задание 31. Символы 7-8
D10484	WORD	Память для хранения названий рецептов. Задание 31. Символы 9-10
D10485	WORD	Память для хранения названий рецептов. Задание 31. Символы 11-12
D10486	WORD	Память для хранения названий рецептов. Задание 31. Символы 13-14
D10487	WORD	Память для хранения названий рецептов. Задание 31. Символы 15-16
D10488	WORD	Память для хранения названий рецептов. Задание 31. Символы 17-18
D10489	WORD	Память для хранения названий рецептов. Задание 31. Символы 19-20
D10490	WORD	Память для хранения названий рецептов. Задание 31. Символы 21-22
D10491	WORD	Память для хранения названий рецептов. Задание 31. Символы 23-24
D10492	WORD	Память для хранения названий рецептов. Задание 31. Символы 25-26
D10493	WORD	Память для хранения названий рецептов. Задание 31. Символы 27-28
D10494	WORD	Память для хранения названий рецептов. Задание 31. Символы 29-30
D10495	WORD	Память для хранения названий рецептов. Задание 31. Символы 31-32
D10496	WORD	Память для хранения названий рецептов. Задание 32. Символы 1-2
D10497	WORD	Память для хранения названий рецептов. Задание 32. Символы 3-4
D10498	WORD	Память для хранения названий рецептов. Задание 32. Символы 5-6
D10499	WORD	Память для хранения названий рецептов. Задание 32. Символы 7-8
D10500	WORD	Память для хранения названий рецептов. Задание 32. Символы 9-10
D10501	WORD	Память для хранения названий рецептов. Задание 32. Символы 11-12
D10502	WORD	Память для хранения названий рецептов. Задание 32. Символы 13-14
D10503	WORD	Память для хранения названий рецептов. Задание 32. Символы 15-16
D10504	WORD	Память для хранения названий рецептов. Задание 32. Символы 17-18
D10505	WORD	Память для хранения названий рецептов. Задание 32. Символы 19-20
D10506	WORD	Память для хранения названий рецептов. Задание 32. Символы 21-22
D10507	WORD	Память для хранения названий рецептов. Задание 32. Символы 23-24
D10508	WORD	Память для хранения названий рецептов. Задание 32. Символы 25-26
D10509	WORD	Память для хранения названий рецептов. Задание 32. Символы 27-28
D10510	WORD	Память для хранения названий рецептов. Задание 32. Символы 29-30
D10511	WORD	Память для хранения названий рецептов. Задание 32. Символы 31-32
D10512	WORD	Память для хранения названий рецептов. Задание 33. Символы 1-2
D10513	WORD	Память для хранения названий рецептов. Задание 33. Символы 3-4
D10514	WORD	Память для хранения названий рецептов. Задание 33. Символы 5-6
D10515	WORD	Память для хранения названий рецептов. Задание 33. Символы 7-8
D10516	WORD	Память для хранения названий рецептов. Задание 33. Символы 9-10
D10517	WORD	Память для хранения названий рецептов. Задание 33. Символы 11-12
D10518	WORD	Память для хранения названий рецептов. Задание 33. Символы 13-14
D10519	WORD	Память для хранения названий рецептов. Задание 33. Символы 15-16
D10520	WORD	Память для хранения названий рецептов. Задание 33. Символы 17-18
D10521	WORD	Память для хранения названий рецептов. Задание 33. Символы 19-20
D10522	WORD	Память для хранения названий рецептов. Задание 33. Символы 21-22
D10523	WORD	Память для хранения названий рецептов. Задание 33. Символы 23-24
D10524	WORD	Память для хранения названий рецептов. Задание 33. Символы 25-26
D10525	WORD	Память для хранения названий рецептов. Задание 33. Символы 27-28
D10526	WORD	Память для хранения названий рецептов. Задание 33. Символы 29-30
D10527	WORD	Память для хранения названий рецептов. Задание 33. Символы 31-32
D10528	WORD	Память для хранения названий рецептов. Задание 34. Символы 1-2
D10529	WORD	Память для хранения названий рецептов. Задание 34. Символы 3-4
D10530	WORD	Память для хранения названий рецептов. Задание 34. Символы 5-6
D10531	WORD	Память для хранения названий рецептов. Задание 34. Символы 7-8
D10532	WORD	Память для хранения названий рецептов. Задание 34. Символы 9-10
D10533	WORD	Память для хранения названий рецептов. Задание 34. Символы 11-12
D10534	WORD	Память для хранения названий рецептов. Задание 34. Символы 13-14
D10535	WORD	Память для хранения названий рецептов. Задание 34. Символы 15-16
D10536	WORD	Память для хранения названий рецептов. Задание 34. Символы 17-18
D10537	WORD	Память для хранения названий рецептов. Задание 34. Символы 19-20
D10538	WORD	Память для хранения названий рецептов. Задание 34. Символы 21-22
D10539	WORD	Память для хранения названий рецептов. Задание 34. Символы 23-24
D10540	WORD	Память для хранения названий рецептов. Задание 34. Символы 25-26
D10541	WORD	Память для хранения названий рецептов. Задание 34. Символы 27-28
D10542	WORD	Память для хранения названий рецептов. Задание 34. Символы 29-30
D10543	WORD	Память для хранения названий рецептов. Задание 34. Символы 31-32
D10544	WORD	Память для хранения названий рецептов. Задание 35. Символы 1-2
D10545	WORD	Память для хранения названий рецептов. Задание 35. Символы 3-4
D10546	WORD	Память для хранения названий рецептов. Задание 35. Символы 5-6
D10547	WORD	Память для хранения названий рецептов. Задание 35. Символы 7-8
D10548	WORD	Память для хранения названий рецептов. Задание 35. Символы 9-10
D10549	WORD	Память для хранения названий рецептов. Задание 35. Символы 11-12
D10550	WORD	Память для хранения названий рецептов. Задание 35. Символы 13-14
D10551	WORD	Память для хранения названий рецептов. Задание 35. Символы 15-16
D10552	WORD	Память для хранения названий рецептов. Задание 35. Символы 17-18
D10553	WORD	Память для хранения названий рецептов. Задание 35. Символы 19-20
D10554	WORD	Память для хранения названий рецептов. Задание 35. Символы 21-22
D10555	WORD	Память для хранения названий рецептов. Задание 35. Символы 23-24
D10556	WORD	Память для хранения названий рецептов. Задание 35. Символы 25-26
D10557	WORD	Память для хранения названий рецептов. Задание 35. Символы 27-28
D10558	WORD	Память для хранения названий рецептов. Задание 35. Символы 29-30
D10559	WORD	Память для хранения названий рецептов. Задание 35. Символы 31-32
D10560	WORD	Память для хранения названий рецептов. Задание 36. Символы 1-2
D10561	WORD	Память для хранения названий рецептов. Задание 36. Символы 3-4
D10562	WORD	Память для хранения названий рецептов. Задание 36. Символы 5-6
D10563	WORD	Память для хранения названий рецептов. Задание 36. Символы 7-8
D10564	WORD	Память для хранения названий рецептов. Задание 36. Символы 9-10
D10565	WORD	Память для хранения названий рецептов. Задание 36. Символы 11-12
D10566	WORD	Память для хранения названий рецептов. Задание 36. Символы 13-14
D10567	WORD	Память для хранения названий рецептов. Задание 36. Символы 15-16
D10568	WORD	Память для хранения названий рецептов. Задание 36. Символы 17-18
D10569	WORD	Память для хранения названий рецептов. Задание 36. Символы 19-20
D10570	WORD	Память для хранения названий рецептов. Задание 36. Символы 21-22
D10571	WORD	Память для хранения названий рецептов. Задание 36. Символы 23-24
D10572	WORD	Память для хранения названий рецептов. Задание 36. Символы 25-26
D10573	WORD	Память для хранения названий рецептов. Задание 36. Символы 27-28
D10574	WORD	Память для хранения названий рецептов. Задание 36. Символы 29-30
D10575	WORD	Память для хранения названий рецептов. Задание 36. Символы 31-32
D10576	WORD	Память для хранения названий рецептов. Задание 37. Символы 1-2
D10577	WORD	Память для хранения названий рецептов. Задание 37. Символы 3-4
D10578	WORD	Память для хранения названий рецептов. Задание 37. Символы 5-6
D10579	WORD	Память для хранения названий рецептов. Задание 37. Символы 7-8
D10580	WORD	Память для хранения названий рецептов. Задание 37. Символы 9-10
D10581	WORD	Память для хранения названий рецептов. Задание 37. Символы 11-12
D10582	WORD	Память для хранения названий рецептов. Задание 37. Символы 13-14
D10583	WORD	Память для хранения названий рецептов. Задание 37. Символы 15-16
D10584	WORD	Память для хранения названий рецептов. Задание 37. Символы 17-18
D10585	WORD	Память для хранения названий рецептов. Задание 37. Символы 19-20
D10586	WORD	Память для хранения названий рецептов. Задание 37. Символы 21-22
D10587	WORD	Память для хранения названий рецептов. Задание 37. Символы 23-24
D10588	WORD	Память для хранения названий рецептов. Задание 37. Символы 25-26
D10589	WORD	Память для хранения названий рецептов. Задание 37. Символы 27-28
D10590	WORD	Память для хранения названий рецептов. Задание 37. Символы 29-30
D10591	WORD	Память для хранения названий рецептов. Задание 37. Символы 31-32
D10592	WORD	Память для хранения названий рецептов. Задание 38. Символы 1-2
D10593	WORD	Память для хранения названий рецептов. Задание 38. Символы 3-4
D10594	WORD	Память для хранения названий рецептов. Задание 38. Символы 5-6
D10595	WORD	Память для хранения названий рецептов. Задание 38. Символы 7-8
D10596	WORD	Память для хранения названий рецептов. Задание 38. Символы 9-10
D10597	WORD	Память для хранения названий рецептов. Задание 38. Символы 11-12
D10598	WORD	Память для хранения названий рецептов. Задание 38. Символы 13-14
D10599	WORD	Память для хранения названий рецептов. Задание 38. Символы 15-16
D10600	WORD	Память для хранения названий рецептов. Задание 38. Символы 17-18
D10601	WORD	Память для хранения названий рецептов. Задание 38. Символы 19-20
D10602	WORD	Память для хранения названий рецептов. Задание 38. Символы 21-22
D10603	WORD	Память для хранения названий рецептов. Задание 38. Символы 23-24
D10604	WORD	Память для хранения названий рецептов. Задание 38. Символы 25-26
D10605	WORD	Память для хранения названий рецептов. Задание 38. Символы 27-28
D10606	WORD	Память для хранения названий рецептов. Задание 38. Символы 29-30
D10607	WORD	Память для хранения названий рецептов. Задание 38. Символы 31-32
D10608	WORD	Память для хранения названий рецептов. Задание 39. Символы 1-2
D10609	WORD	Память для хранения названий рецептов. Задание 39. Символы 3-4
D10610	WORD	Память для хранения названий рецептов. Задание 39. Символы 5-6
D10611	WORD	Память для хранения названий рецептов. Задание 39. Символы 7-8
D10612	WORD	Память для хранения названий рецептов. Задание 39. Символы 9-10
D10613	WORD	Память для хранения названий рецептов. Задание 39. Символы 11-12
D10614	WORD	Память для хранения названий рецептов. Задание 39. Символы 13-14
D10615	WORD	Память для хранения названий рецептов. Задание 39. Символы 15-16
D10616	WORD	Память для хранения названий рецептов. Задание 39. Символы 17-18
D10617	WORD	Память для хранения названий рецептов. Задание 39. Символы 19-20
D10618	WORD	Память для хранения названий рецептов. Задание 39. Символы 21-22
D10619	WORD	Память для хранения названий рецептов. Задание 39. Символы 23-24
D10620	WORD	Память для хранения названий рецептов. Задание 39. Символы 25-26
D10621	WORD	Память для хранения названий рецептов. Задание 39. Символы 27-28
D10622	WORD	Память для хранения названий рецептов. Задание 39. Символы 29-30
D10623	WORD	Память для хранения названий рецептов. Задание 39. Символы 31-32
D10624	WORD	Память для хранения названий рецептов. Задание 40. Символы 1-2
D10625	WORD	Память для хранения названий рецептов. Задание 40. Символы 3-4
D10626	WORD	Память для хранения названий рецептов. Задание 40. Символы 5-6
D10627	WORD	Память для хранения названий рецептов. Задание 40. Символы 7-8
D10628	WORD	Память для хранения названий рецептов. Задание 40. Символы 9-10
D10629	WORD	Память для хранения названий рецептов. Задание 40. Символы 11-12
D10630	WORD	Память для хранения названий рецептов. Задание 40. Символы 13-14
D10631	WORD	Память для хранения названий рецептов. Задание 40. Символы 15-16
D10632	WORD	Память для хранения названий рецептов. Задание 40. Символы 17-18
D10633	WORD	Память для хранения названий рецептов. Задание 40. Символы 19-20
D10634	WORD	Память для хранения названий рецептов. Задание 40. Символы 21-22
D10635	WORD	Память для хранения названий рецептов. Задание 40. Символы 23-24
D10636	WORD	Память для хранения названий рецептов. Задание 40. Символы 25-26
D10637	WORD	Память для хранения названий рецептов. Задание 40. Символы 27-28
D10638	WORD	Память для хранения названий рецептов. Задание 40. Символы 29-30
D10639	WORD	Память для хранения названий рецептов. Задание 40. Символы 31-32
D10640	WORD	Память для хранения названий рецептов. Задание 41. Символы 1-2
D10641	WORD	Память для хранения названий рецептов. Задание 41. Символы 3-4
D10642	WORD	Память для хранения названий рецептов. Задание 41. Символы 5-6
D10643	WORD	Память для хранения названий рецептов. Задание 41. Символы 7-8
D10644	WORD	Память для хранения названий рецептов. Задание 41. Символы 9-10
D10645	WORD	Память для хранения названий рецептов. Задание 41. Символы 11-12
D10646	WORD	Память для хранения названий рецептов. Задание 41. Символы 13-14
D10647	WORD	Память для хранения названий рецептов. Задание 41. Символы 15-16
D10648	WORD	Память для хранения названий рецептов. Задание 41. Символы 17-18
D10649	WORD	Память для хранения названий рецептов. Задание 41. Символы 19-20
D10650	WORD	Память для хранения названий рецептов. Задание 41. Символы 21-22
D10651	WORD	Память для хранения названий рецептов. Задание 41. Символы 23-24
D10652	WORD	Память для хранения названий рецептов. Задание 41. Символы 25-26
D10653	WORD	Память для хранения названий рецептов. Задание 41. Символы 27-28
D10654	WORD	Память для хранения названий рецептов. Задание 41. Символы 29-30
D10655	WORD	Память для хранения названий рецептов. Задание 41. Символы 31-32
D10656	WORD	Память для хранения названий рецептов. Задание 42. Символы 1-2
D10657	WORD	Память для хранения названий рецептов. Задание 42. Символы 3-4
D10658	WORD	Память для хранения названий рецептов. Задание 42. Символы 5-6
D10659	WORD	Память для хранения названий рецептов. Задание 42. Символы 7-8
D10660	WORD	Память для хранения названий рецептов. Задание 42. Символы 9-10
D10661	WORD	Память для хранения названий рецептов. Задание 42. Символы 11-12
D10662	WORD	Память для хранения названий рецептов. Задание 42. Символы 13-14
D10663	WORD	Память для хранения названий рецептов. Задание 42. Символы 15-16
D10664	WORD	Память для хранения названий рецептов. Задание 42. Символы 17-18
D10665	WORD	Память для хранения названий рецептов. Задание 42. Символы 19-20
D10666	WORD	Память для хранения названий рецептов. Задание 42. Символы 21-22
D10667	WORD	Память для хранения названий рецептов. Задание 42. Символы 23-24
D10668	WORD	Память для хранения названий рецептов. Задание 42. Символы 25-26
D10669	WORD	Память для хранения названий рецептов. Задание 42. Символы 27-28
D10670	WORD	Память для хранения названий рецептов. Задание 42. Символы 29-30
D10671	WORD	Память для хранения названий рецептов. Задание 42. Символы 31-32
D10672	WORD	Память для хранения названий рецептов. Задание 43. Символы 1-2
D10673	WORD	Память для хранения названий рецептов. Задание 43. Символы 3-4
D10674	WORD	Память для хранения названий рецептов. Задание 43. Символы 5-6
D10675	WORD	Память для хранения названий рецептов. Задание 43. Символы 7-8
D10676	WORD	Память для хранения названий рецептов. Задание 43. Символы 9-10
D10677	WORD	Память для хранения названий рецептов. Задание 43. Символы 11-12
D10678	WORD	Память для хранения названий рецептов. Задание 43. Символы 13-14
D10679	WORD	Память для хранения названий рецептов. Задание 43. Символы 15-16
D10680	WORD	Память для хранения названий рецептов. Задание 43. Символы 17-18
D10681	WORD	Память для хранения названий рецептов. Задание 43. Символы 19-20
D10682	WORD	Память для хранения названий рецептов. Задание 43. Символы 21-22
D10683	WORD	Память для хранения названий рецептов. Задание 43. Символы 23-24
D10684	WORD	Память для хранения названий рецептов. Задание 43. Символы 25-26
D10685	WORD	Память для хранения названий рецептов. Задание 43. Символы 27-28
D10686	WORD	Память для хранения названий рецептов. Задание 43. Символы 29-30
D10687	WORD	Память для хранения названий рецептов. Задание 43. Символы 31-32
D10688	WORD	Память для хранения названий рецептов. Задание 44. Символы 1-2
D10689	WORD	Память для хранения названий рецептов. Задание 44. Символы 3-4
D10690	WORD	Память для хранения названий рецептов. Задание 44. Символы 5-6
D10691	WORD	Память для хранения названий рецептов. Задание 44. Символы 7-8
D10692	WORD	Память для хранения названий рецептов. Задание 44. Символы 9-10
D10693	WORD	Память для хранения названий рецептов. Задание 44. Символы 11-12
D10694	WORD	Память для хранения названий рецептов. Задание 44. Символы 13-14
D10695	WORD	Память для хранения названий рецептов. Задание 44. Символы 15-16
D10696	WORD	Память для хранения названий рецептов. Задание 44. Символы 17-18
D10697	WORD	Память для хранения названий рецептов. Задание 44. Символы 19-20
D10698	WORD	Память для хранения названий рецептов. Задание 44. Символы 21-22
D10699	WORD	Память для хранения названий рецептов. Задание 44. Символы 23-24
D10700	WORD	Память для хранения названий рецептов. Задание 44. Символы 25-26
D10701	WORD	Память для хранения названий рецептов. Задание 44. Символы 27-28
D10702	WORD	Память для хранения названий рецептов. Задание 44. Символы 29-30
D10703	WORD	Память для хранения названий рецептов. Задание 44. Символы 31-32
D10704	WORD	Память для хранения названий рецептов. Задание 45. Символы 1-2
D10705	WORD	Память для хранения названий рецептов. Задание 45. Символы 3-4
D10706	WORD	Память для хранения названий рецептов. Задание 45. Символы 5-6
D10707	WORD	Память для хранения названий рецептов. Задание 45. Символы 7-8
D10708	WORD	Память для хранения названий рецептов. Задание 45. Символы 9-10
D10709	WORD	Память для хранения названий рецептов. Задание 45. Символы 11-12
D10710	WORD	Память для хранения названий рецептов. Задание 45. Символы 13-14
D10711	WORD	Память для хранения названий рецептов. Задание 45. Символы 15-16
D10712	WORD	Память для хранения названий рецептов. Задание 45. Символы 17-18
D10713	WORD	Память для хранения названий рецептов. Задание 45. Символы 19-20
D10714	WORD	Память для хранения названий рецептов. Задание 45. Символы 21-22
D10715	WORD	Память для хранения названий рецептов. Задание 45. Символы 23-24
D10716	WORD	Память для хранения названий рецептов. Задание 45. Символы 25-26
D10717	WORD	Память для хранения названий рецептов. Задание 45. Символы 27-28
D10718	WORD	Память для хранения названий рецептов. Задание 45. Символы 29-30
D10719	WORD	Память для хранения названий рецептов. Задание 45. Символы 31-32
D10720	WORD	Память для хранения названий рецептов. Задание 46. Символы 1-2
D10721	WORD	Память для хранения названий рецептов. Задание 46. Символы 3-4
D10722	WORD	Память для хранения названий рецептов. Задание 46. Символы 5-6
D10723	WORD	Память для хранения названий рецептов. Задание 46. Символы 7-8
D10724	WORD	Память для хранения названий рецептов. Задание 46. Символы 9-10
D10725	WORD	Память для хранения названий рецептов. Задание 46. Символы 11-12
D10726	WORD	Память для хранения названий рецептов. Задание 46. Символы 13-14
D10727	WORD	Память для хранения названий рецептов. Задание 46. Символы 15-16
D10728	WORD	Память для хранения названий рецептов. Задание 46. Символы 17-18
D10729	WORD	Память для хранения названий рецептов. Задание 46. Символы 19-20
D10730	WORD	Память для хранения названий рецептов. Задание 46. Символы 21-22
D10731	WORD	Память для хранения названий рецептов. Задание 46. Символы 23-24
D10732	WORD	Память для хранения названий рецептов. Задание 46. Символы 25-26
D10733	WORD	Память для хранения названий рецептов. Задание 46. Символы 27-28
D10734	WORD	Память для хранения названий рецептов. Задание 46. Символы 29-30
D10735	WORD	Память для хранения названий рецептов. Задание 46. Символы 31-32
D10736	WORD	Память для хранения названий рецептов. Задание 47. Символы 1-2
D10737	WORD	Память для хранения названий рецептов. Задание 47. Символы 3-4
D10738	WORD	Память для хранения названий рецептов. Задание 47. Символы 5-6
D10739	WORD	Память для хранения названий рецептов. Задание 47. Символы 7-8
D10740	WORD	Память для хранения названий рецептов. Задание 47. Символы 9-10
D10741	WORD	Память для хранения названий рецептов. Задание 47. Символы 11-12
D10742	WORD	Память для хранения названий рецептов. Задание 47. Символы 13-14
D10743	WORD	Память для хранения названий рецептов. Задание 47. Символы 15-16
D10744	WORD	Память для хранения названий рецептов. Задание 47. Символы 17-18
D10745	WORD	Память для хранения названий рецептов. Задание 47. Символы 19-20
D10746	WORD	Память для хранения названий рецептов. Задание 47. Символы 21-22
D10747	WORD	Память для хранения названий рецептов. Задание 47. Символы 23-24
D10748	WORD	Память для хранения названий рецептов. Задание 47. Символы 25-26
D10749	WORD	Память для хранения названий рецептов. Задание 47. Символы 27-28
D10750	WORD	Память для хранения названий рецептов. Задание 47. Символы 29-30
D10751	WORD	Память для хранения названий рецептов. Задание 47. Символы 31-32
D10752	WORD	Память для хранения названий рецептов. Задание 48. Символы 1-2
D10753	WORD	Память для хранения названий рецептов. Задание 48. Символы 3-4
D10754	WORD	Память для хранения названий рецептов. Задание 48. Символы 5-6
D10755	WORD	Память для хранения названий рецептов. Задание 48. Символы 7-8
D10756	WORD	Память для хранения названий рецептов. Задание 48. Символы 9-10
D10757	WORD	Память для хранения названий рецептов. Задание 48. Символы 11-12
D10758	WORD	Память для хранения названий рецептов. Задание 48. Символы 13-14
D10759	WORD	Память для хранения названий рецептов. Задание 48. Символы 15-16
D10760	WORD	Память для хранения названий рецептов. Задание 48. Символы 17-18
D10761	WORD	Память для хранения названий рецептов. Задание 48. Символы 19-20
D10762	WORD	Память для хранения названий рецептов. Задание 48. Символы 21-22
D10763	WORD	Память для хранения названий рецептов. Задание 48. Символы 23-24
D10764	WORD	Память для хранения названий рецептов. Задание 48. Символы 25-26
D10765	WORD	Память для хранения названий рецептов. Задание 48. Символы 27-28
D10766	WORD	Память для хранения названий рецептов. Задание 48. Символы 29-30
D10767	WORD	Память для хранения названий рецептов. Задание 48. Символы 31-32
D10768	WORD	Память для хранения названий рецептов. Задание 49. Символы 1-2
D10769	WORD	Память для хранения названий рецептов. Задание 49. Символы 3-4
D10770	WORD	Память для хранения названий рецептов. Задание 49. Символы 5-6
D10771	WORD	Память для хранения названий рецептов. Задание 49. Символы 7-8
D10772	WORD	Память для хранения названий рецептов. Задание 49. Символы 9-10
D10773	WORD	Память для хранения названий рецептов. Задание 49. Символы 11-12
D10774	WORD	Память для хранения названий рецептов. Задание 49. Символы 13-14
D10775	WORD	Память для хранения названий рецептов. Задание 49. Символы 15-16
D10776	WORD	Память для хранения названий рецептов. Задание 49. Символы 17-18
D10777	WORD	Память для хранения названий рецептов. Задание 49. Символы 19-20
D10778	WORD	Память для хранения названий рецептов. Задание 49. Символы 21-22
D10779	WORD	Память для хранения названий рецептов. Задание 49. Символы 23-24
D10780	WORD	Память для хранения названий рецептов. Задание 49. Символы 25-26
D10781	WORD	Память для хранения названий рецептов. Задание 49. Символы 27-28
D10782	WORD	Память для хранения названий рецептов. Задание 49. Символы 29-30
D10783	WORD	Память для хранения названий рецептов. Задание 49. Символы 31-32
D10784	WORD	Память для хранения названий рецептов. Задание 50. Символы 1-2
D10785	WORD	Память для хранения названий рецептов. Задание 50. Символы 3-4
D10786	WORD	Память для хранения названий рецептов. Задание 50. Символы 5-6
D10787	WORD	Память для хранения названий рецептов. Задание 50. Символы 7-8
D10788	WORD	Память для хранения названий рецептов. Задание 50. Символы 9-10
D10789	WORD	Память для хранения названий рецептов. Задание 50. Символы 11-12
D10790	WORD	Память для хранения названий рецептов. Задание 50. Символы 13-14
D10791	WORD	Память для хранения названий рецептов. Задание 50. Символы 15-16
D10792	WORD	Память для хранения названий рецептов. Задание 50. Символы 17-18
D10793	WORD	Память для хранения названий рецептов. Задание 50. Символы 19-20
D10794	WORD	Память для хранения названий рецептов. Задание 50. Символы 21-22
D10795	WORD	Память для хранения названий рецептов. Задание 50. Символы 23-24
D10796	WORD	Память для хранения названий рецептов. Задание 50. Символы 25-26
D10797	WORD	Память для хранения названий рецептов. Задание 50. Символы 27-28
D10798	WORD	Память для хранения названий рецептов. Задание 50. Символы 29-30
D10799	WORD	Память для хранения названий рецептов. Задание 50. Символы 31-32
D10800	WORD	Память для хранения названий рецептов. Задание 51. Символы 1-2
D10801	WORD	Память для хранения названий рецептов. Задание 51. Символы 3-4
D10802	WORD	Память для хранения названий рецептов. Задание 51. Символы 5-6
D10803	WORD	Память для хранения названий рецептов. Задание 51. Символы 7-8
D10804	WORD	Память для хранения названий рецептов. Задание 51. Символы 9-10
D10805	WORD	Память для хранения названий рецептов. Задание 51. Символы 11-12
D10806	WORD	Память для хранения названий рецептов. Задание 51. Символы 13-14
D10807	WORD	Память для хранения названий рецептов. Задание 51. Символы 15-16
D10808	WORD	Память для хранения названий рецептов. Задание 51. Символы 17-18
D10809	WORD	Память для хранения названий рецептов. Задание 51. Символы 19-20
D10810	WORD	Память для хранения названий рецептов. Задание 51. Символы 21-22
D10811	WORD	Память для хранения названий рецептов. Задание 51. Символы 23-24
D10812	WORD	Память для хранения названий рецептов. Задание 51. Символы 25-26
D10813	WORD	Память для хранения названий рецептов. Задание 51. Символы 27-28
D10814	WORD	Память для хранения названий рецептов. Задание 51. Символы 29-30
D10815	WORD	Память для хранения названий рецептов. Задание 51. Символы 31-32
D10816	WORD	Память для хранения названий рецептов. Задание 52. Символы 1-2
D10817	WORD	Память для хранения названий рецептов. Задание 52. Символы 3-4
D10818	WORD	Память для хранения названий рецептов. Задание 52. Символы 5-6
D10819	WORD	Память для хранения названий рецептов. Задание 52. Символы 7-8
D10820	WORD	Память для хранения названий рецептов. Задание 52. Символы 9-10
D10821	WORD	Память для хранения названий рецептов. Задание 52. Символы 11-12
D10822	WORD	Память для хранения названий рецептов. Задание 52. Символы 13-14
D10823	WORD	Память для хранения названий рецептов. Задание 52. Символы 15-16
D10824	WORD	Память для хранения названий рецептов. Задание 52. Символы 17-18
D10825	WORD	Память для хранения названий рецептов. Задание 52. Символы 19-20
D10826	WORD	Память для хранения названий рецептов. Задание 52. Символы 21-22
D10827	WORD	Память для хранения названий рецептов. Задание 52. Символы 23-24
D10828	WORD	Память для хранения названий рецептов. Задание 52. Символы 25-26
D10829	WORD	Память для хранения названий рецептов. Задание 52. Символы 27-28
D10830	WORD	Память для хранения названий рецептов. Задание 52. Символы 29-30
D10831	WORD	Память для хранения названий рецептов. Задание 52. Символы 31-32
D10832	WORD	Память для хранения названий рецептов. Задание 53. Символы 1-2
D10833	WORD	Память для хранения названий рецептов. Задание 53. Символы 3-4
D10834	WORD	Память для хранения названий рецептов. Задание 53. Символы 5-6
D10835	WORD	Память для хранения названий рецептов. Задание 53. Символы 7-8
D10836	WORD	Память для хранения названий рецептов. Задание 53. Символы 9-10
D10837	WORD	Память для хранения названий рецептов. Задание 53. Символы 11-12
D10838	WORD	Память для хранения названий рецептов. Задание 53. Символы 13-14
D10839	WORD	Память для хранения названий рецептов. Задание 53. Символы 15-16
D10840	WORD	Память для хранения названий рецептов. Задание 53. Символы 17-18
D10841	WORD	Память для хранения названий рецептов. Задание 53. Символы 19-20
D10842	WORD	Память для хранения названий рецептов. Задание 53. Символы 21-22
D10843	WORD	Память для хранения названий рецептов. Задание 53. Символы 23-24
D10844	WORD	Память для хранения названий рецептов. Задание 53. Символы 25-26
D10845	WORD	Память для хранения названий рецептов. Задание 53. Символы 27-28
D10846	WORD	Память для хранения названий рецептов. Задание 53. Символы 29-30
D10847	WORD	Память для хранения названий рецептов. Задание 53. Символы 31-32
D10848	WORD	Память для хранения названий рецептов. Задание 54. Символы 1-2
D10849	WORD	Память для хранения названий рецептов. Задание 54. Символы 3-4
D10850	WORD	Память для хранения названий рецептов. Задание 54. Символы 5-6
D10851	WORD	Память для хранения названий рецептов. Задание 54. Символы 7-8
